LIN {X 0,Y 268.905,Z 288.913,A -85,B 0,C 180,E1 -18635.456,E2 -18635.456} C_VEL
LIN {X 0,Y 261.932,Z 271.443,A -85,B 0,C 180,E1 -18636.717,E2 -18636.717} C_VEL
LIN {X 0,Y 257.784,Z 261.083,A -85,B 0,C 180,E1 -18637.566,E2 -18637.566} C_VEL
LIN {X 0,Y 256.379,Z 255.314,A -85,B 0,C 180,E1 -18639.936,E2 -18639.936} C_VEL
LIN {X 0,Y 256.266,Z 255.064,A -85,B 0,C 180,E1 -18641.069,E2 -18641.069} C_VEL
LIN {X 0,Y 256.221,Z 255.067,A -85,B 0,C 180,E1 -18644.293,E2 -18644.293} C_VEL
LIN {X 0,Y 256.173,Z 255.073,A -85,B 0,C 180,E1 -18647.566,E2 -18647.566} C_VEL
LIN {X 0,Y 256.113,Z 255.08,A -85,B 0,C 180,E1 -18651.113,E2 -18651.113} C_VEL
LIN {X 0,Y 256.105,Z 255.077,A -85,B 0,C 180,E1 -18655.115,E2 -18655.115} C_VEL
LIN {X 0,Y 256.017,Z 255.078,A -85,B 0,C 180,E1 -18659.613,E2 -18659.613} C_VEL
LIN {X 0,Y 256.041,Z 255.087,A -85,B 0,C 180,E1 -18663.298,E2 -18663.298} C_VEL
LIN {X 0,Y 256.094,Z 255.082,A -85,B 0,C 180,E1 -18667.276,E2 -18667.276} C_VEL
LIN {X 0,Y 255.996,Z 255.082,A -85,B 0,C 180,E1 -18671.216,E2 -18671.216} C_VEL
LIN {X 0,Y 255.998,Z 255.094,A -85,B 0,C 180,E1 -18675.545,E2 -18675.545} C_VEL
LIN {X 0,Y 256,Z 255.085,A -85,B 0,C 180,E1 -18678.795,E2 -18678.795} C_VEL
LIN {X 0,Y 256.087,Z 255.063,A -85,B 0,C 180,E1 -18682.868,E2 -18682.868} C_VEL
LIN {X 0,Y 256.053,Z 255.09,A -85,B 0,C 180,E1 -18686.713,E2 -18686.713} C_VEL
LIN {X 0,Y 256.029,Z 255.058,A -85,B 0,C 180,E1 -18690.397,E2 -18690.397} C_VEL
LIN {X 0,Y 256.057,Z 255.074,A -85,B 0,C 180,E1 -18693.957,E2 -18693.957} C_VEL
LIN {X 0,Y 256.055,Z 255.089,A -85,B 0,C 180,E1 -18697.409,E2 -18697.409} C_VEL
LIN {X 0,Y 256.148,Z 255.047,A -85,B 0,C 180,E1 -18700.783,E2 -18700.783} C_VEL
LIN {X 0,Y 256.241,Z 255.032,A -85,B 0,C 180,E1 -18704.087,E2 -18704.087} C_VEL
LIN {X 0,Y 256.284,Z 255.057,A -85,B 0,C 180,E1 -18707.333,E2 -18707.333} C_VEL
LIN {X 0,Y 256.434,Z 255.031,A -85,B 0,C 180,E1 -18710.628,E2 -18710.628} C_VEL
LIN {X 0,Y 256.382,Z 255.005,A -85,B 0,C 180,E1 -18714.228,E2 -18714.228} C_VEL
LIN {X 0,Y 256.698,Z 255.005,A -85,B 0,C 180,E1 -18718.437,E2 -18718.437} C_VEL
LIN {X 0,Y 256.68,Z 255.005,A -85,B 0,C 180,E1 -18721.093,E2 -18721.093} C_VEL
LIN {X 0,Y 256.371,Z 255.041,A -85,B 0,C 180,E1 -18721.967,E2 -18721.967} C_VEL
LIN {X 0,Y 254.985,Z 255.205,A -85,B 0,C 180,E1 -18723.254,E2 -18723.254} C_VEL
LIN {X 0,Y 250.536,Z 255.744,A -85,B 0,C 180,E1 -18726.253,E2 -18726.253} C_VEL
LIN {X 0,Y 249.504,Z 255.89,A -85,B 0,C 180,E1 -18727.599,E2 -18727.599} C_VEL
LIN {X 0,Y 249.444,Z 255.899,A -85,B 0,C 180,E1 -18728.055,E2 -18728.055} C_VEL
LIN {X 0,Y 249.25,Z 255.935,A -85,B 0,C 180,E1 -18731.389,E2 -18731.389} C_VEL
LIN {X 0,Y 249.206,Z 255.915,A -85,B 0,C 180,E1 -18736.386,E2 -18736.386} C_VEL
LIN {X 0,Y 249.091,Z 255.95,A -85,B 0,C 180,E1 -18741.523,E2 -18741.523} C_VEL
LIN {X 0,Y 249.097,Z 255.938,A -85,B 0,C 180,E1 -18745.463,E2 -18745.463} C_VEL
LIN {X 0,Y 249.05,Z 255.959,A -85,B 0,C 180,E1 -18748.977,E2 -18748.977} C_VEL
LIN {X 0,Y 249.041,Z 255.95,A -85,B 0,C 180,E1 -18752.43,E2 -18752.43} C_VEL
LIN {X 0,Y 249.027,Z 255.956,A -85,B 0,C 180,E1 -18756.351,E2 -18756.351} C_VEL
LIN {X 0,Y 248.993,Z 255.969,A -85,B 0,C 180,E1 -18760.486,E2 -18760.486} C_VEL
LIN {X 0,Y 248.977,Z 255.972,A -85,B 0,C 180,E1 -18764.891,E2 -18764.891} C_VEL
LIN {X 0,Y 249.008,Z 255.964,A -85,B 0,C 180,E1 -18767.36,E2 -18767.36} C_VEL
LIN {X 0,Y 249.059,Z 255.959,A -85,B 0,C 180,E1 -18772.202,E2 -18772.202} C_VEL
LIN {X 0,Y 249.104,Z 255.988,A -85,B 0,C 180,E1 -18774.006,E2 -18774.006} C_VEL
LIN {X 0,Y 249.603,Z 258.24,A -85,B 0,C 180,E1 -18775.097,E2 -18775.097} C_VEL
LIN {X 0,Y 251.579,Z 267.236,A -85,B 0,C 180,E1 -18778.731,E2 -18778.731} C_VEL
LIN {X 0,Y 257.031,Z 280.617,A -85,B 0,C 180,E1 -18779.858,E2 -18779.858} C_VEL
LIN {X 0,Y 260.891,Z 291.121,A -85,B 0,C 180,E1 -18780.616,E2 -18780.616} C_VEL
LIN {X 0,Y 264.281,Z 312.794,A -85,B 0,C 180,E1 -18781.64,E2 -18781.64} C_VEL
LIN {X 0,Y 262.135,Z 374.903,A -85,B 0,C 180,E1 -18783.368,E2 -18783.368} C_VEL
LIN {X 0,Y 261.159,Z 388.066,A -85,B 0,C 180,E1 -18784.014,E2 -18784.014} C_VEL
LIN {X 0,Y 259.679,Z 401.335,A -85,B 0,C 180,E1 -18784.982,E2 -18784.982} C_VEL
LIN {X 0,Y 258.161,Z 412.517,A -85,B 0,C 180,E1 -18786.111,E2 -18786.111} C_VEL
LIN {X 0,Y 256.245,Z 424.145,A -85,B 0,C 180,E1 -18787.631,E2 -18787.631} C_VEL
LIN {X 0,Y 254.349,Z 434.623,A -85,B 0,C 180,E1 -18789.371,E2 -18789.371} C_VEL
LIN {X 0,Y 252.494,Z 444.866,A -85,B 0,C 180,E1 -18791.54,E2 -18791.54} C_VEL
LIN {X 0,Y 250.791,Z 453.135,A -85,B 0,C 180,E1 -18793.725,E2 -18793.725} C_VEL
LIN {X 0,Y 249.263,Z 460.448,A -85,B 0,C 180,E1 -18796.132,E2 -18796.132} C_VEL
LIN {X 0,Y 248.217,Z 466.292,A -85,B 0,C 180,E1 -18798.567,E2 -18798.567} C_VEL
LIN {X 0,Y 247.494,Z 470.875,A -85,B 0,C 180,E1 -18801.013,E2 -18801.013} C_VEL
LIN {X 0,Y 247.038,Z 474.348,A -85,B 0,C 180,E1 -18803.464,E2 -18803.464} C_VEL
LIN {X 0,Y 246.882,Z 476.113,A -85,B 0,C 180,E1 -18805.143,E2 -18805.143} C_VEL
LIN {X 0,Y 246.866,Z 478.303,A -85,B 0,C 180,E1 -18808.367,E2 -18808.367} C_VEL
LIN {X 0,Y 246.9,Z 478.807,A -85,B 0,C 180,E1 -18809.999,E2 -18809.999} C_VEL
LIN {X 0,Y 246.867,Z 478.878,A -85,B 0,C 180,E1 -18811.63,E2 -18811.63} C_VEL
LIN {X 0,Y 246.897,Z 477.862,A -85,B 0,C 180,E1 -18814.897,E2 -18814.897} C_VEL
LIN {X 0,Y 247.097,Z 476.762,A -85,B 0,C 180,E1 -18816.531,E2 -18816.531} C_VEL
LIN {X 0,Y 247.385,Z 475.213,A -85,B 0,C 180,E1 -18818.165,E2 -18818.165} C_VEL
LIN {X 0,Y 248.065,Z 472.112,A -85,B 0,C 180,E1 -18820.61,E2 -18820.61} C_VEL
LIN {X 0,Y 249.118,Z 467.968,A -85,B 0,C 180,E1 -18823.042,E2 -18823.042} C_VEL
LIN {X 0,Y 250.567,Z 462.667,A -85,B 0,C 180,E1 -18825.452,E2 -18825.452} C_VEL
LIN {X 0,Y 252.492,Z 456.034,A -85,B 0,C 180,E1 -18827.828,E2 -18827.828} C_VEL
LIN {X 0,Y 254.765,Z 447.424,A -85,B 0,C 180,E1 -18830.283,E2 -18830.283} C_VEL
LIN {X 0,Y 256.764,Z 439.438,A -85,B 0,C 180,E1 -18832.107,E2 -18832.107} C_VEL
LIN {X 0,Y 259.312,Z 429.101,A -85,B 0,C 180,E1 -18833.986,E2 -18833.986} C_VEL
LIN {X 0,Y 261.853,Z 417.489,A -85,B 0,C 180,E1 -18835.643,E2 -18835.643} C_VEL
LIN {X 0,Y 263.96,Z 405.99,A -85,B 0,C 180,E1 -18836.911,E2 -18836.911} C_VEL
LIN {X 0,Y 265.877,Z 392.843,A -85,B 0,C 180,E1 -18837.98,E2 -18837.98} C_VEL
LIN {X 0,Y 267.225,Z 380.531,A -85,B 0,C 180,E1 -18838.68,E2 -18838.68} C_VEL
LIN {X 0,Y 268.125,Z 367.233,A -85,B 0,C 180,E1 -18839.145,E2 -18839.145} C_VEL
LIN {X 0,Y 270.109,Z 314.39,A -85,B 0,C 180,E1 -18840.605,E2 -18840.605} C_VEL
LIN {X 0,Y 267.568,Z 298.937,A -85,B 0,C 180,E1 -18841.502,E2 -18841.502} C_VEL
LIN {X 0,Y 261.325,Z 284.682,A -85,B 0,C 180,E1 -18842.985,E2 -18842.985} C_VEL
LIN {X 0,Y 254.135,Z 270.585,A -85,B 0,C 180,E1 -18844.756,E2 -18844.756} C_VEL
LIN {X 0,Y 251.849,Z 266.387,A -85,B 0,C 180,E1 -18845.407,E2 -18845.407} C_VEL
LIN {X 0,Y 250.675,Z 261.826,A -85,B 0,C 180,E1 -18847.445,E2 -18847.445} C_VEL
LIN {X 0,Y 248.999,Z 256.011,A -85,B 0,C 180,E1 -18850.51,E2 -18850.51} C_VEL
LIN {X 0,Y 248.969,Z 255.972,A -85,B 0,C 180,E1 -18854.885,E2 -18854.885} C_VEL
LIN {X 0,Y 248.985,Z 255.971,A -85,B 0,C 180,E1 -18857.351,E2 -18857.351} C_VEL
LIN {X 0,Y 249.048,Z 255.957,A -85,B 0,C 180,E1 -18862.196,E2 -18862.196} C_VEL
LIN {X 0,Y 249.047,Z 255.957,A -85,B 0,C 180,E1 -18865.635,E2 -18865.635} C_VEL
LIN {X 0,Y 249.005,Z 255.962,A -85,B 0,C 180,E1 -18869.462,E2 -18869.462} C_VEL
LIN {X 0,Y 249.036,Z 255.954,A -85,B 0,C 180,E1 -18873.153,E2 -18873.153} C_VEL
LIN {X 0,Y 249.054,Z 255.95,A -85,B 0,C 180,E1 -18876.725,E2 -18876.725} C_VEL
LIN {X 0,Y 249.09,Z 255.955,A -85,B 0,C 180,E1 -18880.205,E2 -18880.205} C_VEL
LIN {X 0,Y 249.195,Z 255.944,A -85,B 0,C 180,E1 -18883.614,E2 -18883.614} C_VEL
LIN {X 0,Y 249.23,Z 255.938,A -85,B 0,C 180,E1 -18888.61,E2 -18888.61} C_VEL
LIN {X 0,Y 249.417,Z 255.903,A -85,B 0,C 180,E1 -18891.895,E2 -18891.895} C_VEL
LIN {X 0,Y 249.25,Z 255.93,A -85,B 0,C 180,E1 -18895.142,E2 -18895.142} C_VEL
LIN {X 0,Y 249.65,Z 255.887,A -85,B 0,C 180,E1 -18898.381,E2 -18898.381} C_VEL
LIN {X 0,Y 249.638,Z 255.877,A -85,B 0,C 180,E1 -18901.608,E2 -18901.608} C_VEL
LIN {X 0,Y 249.411,Z 255.909,A -85,B 0,C 180,E1 -18906.554,E2 -18906.554} C_VEL
LIN {X 0,Y 249.331,Z 255.918,A -85,B 0,C 180,E1 -18909.731,E2 -18909.731} C_VEL
LIN {X 0,Y 249.164,Z 255.947,A -85,B 0,C 180,E1 -18914.7,E2 -18914.7} C_VEL
LIN {X 0,Y 249.099,Z 255.954,A -85,B 0,C 180,E1 -18918.074,E2 -18918.074} C_VEL
LIN {X 0,Y 249.064,Z 255.962,A -85,B 0,C 180,E1 -18921.514,E2 -18921.514} C_VEL
LIN {X 0,Y 249.066,Z 255.957,A -85,B 0,C 180,E1 -18925.455,E2 -18925.455} C_VEL
LIN {X 0,Y 249.06,Z 256.056,A -85,B 0,C 180,E1 -18928.815,E2 -18928.815} C_VEL
LIN {X 0,Y 250.411,Z 261.075,A -85,B 0,C 180,E1 -18931.331,E2 -18931.331} C_VEL
LIN {X 0,Y 252.768,Z 265.242,A -85,B 0,C 180,E1 -18932.036,E2 -18932.036} C_VEL
LIN {X 0,Y 260.17,Z 278.693,A -85,B 0,C 180,E1 -18933.851,E2 -18933.851} C_VEL
LIN {X 0,Y 266.998,Z 293.384,A -85,B 0,C 180,E1 -18935.466,E2 -18935.466} C_VEL
LIN {X 0,Y 270.294,Z 301.89,A -85,B 0,C 180,E1 -18936.249,E2 -18936.249} C_VEL
LIN {X 0,Y 270.478,Z 305.292,A -85,B 0,C 180,E1 -18936.39,E2 -18936.39} C_VEL
LIN {X 0,Y 267.773,Z 368.475,A -85,B 0,C 180,E1 -18938.132,E2 -18938.132} C_VEL
LIN {X 0,Y 266.626,Z 381.328,A -85,B 0,C 180,E1 -18938.741,E2 -18938.741} C_VEL
LIN {X 0,Y 265.179,Z 393.57,A -85,B 0,C 180,E1 -18939.614,E2 -18939.614} C_VEL
LIN {X 0,Y 263.303,Z 405.552,A -85,B 0,C 180,E1 -18940.769,E2 -18940.769} C_VEL
LIN {X 0,Y 260.997,Z 417.533,A -85,B 0,C 180,E1 -18942.305,E2 -18942.305} C_VEL
LIN {X 0,Y 258.672,Z 427.674,A -85,B 0,C 180,E1 -18943.948,E2 -18943.948} C_VEL
LIN {X 0,Y 256.398,Z 436.734,A -85,B 0,C 180,E1 -18945.78,E2 -18945.78} C_VEL
LIN {X 0,Y 254.141,Z 445.083,A -85,B 0,C 180,E1 -18947.888,E2 -18947.888} C_VEL
LIN {X 0,Y 252.228,Z 452.224,A -85,B 0,C 180,E1 -18950.146,E2 -18950.146} C_VEL
LIN {X 0,Y 250.271,Z 459.008,A -85,B 0,C 180,E1 -18952.863,E2 -18952.863} C_VEL
LIN {X 0,Y 248.792,Z 464.189,A -85,B 0,C 180,E1 -18955.602,E2 -18955.602} C_VEL
LIN {X 0,Y 247.8,Z 467.877,A -85,B 0,C 180,E1 -18958.29,E2 -18958.29} C_VEL
LIN {X 0,Y 247.073,Z 470.447,A -85,B 0,C 180,E1 -18961.083,E2 -18961.083} C_VEL
LIN {X 0,Y 246.731,Z 471.477,A -85,B 0,C 180,E1 -18962.888,E2 -18962.888} C_VEL
LIN {X 0,Y 246.46,Z 472.111,A -85,B 0,C 180,E1 -18965.836,E2 -18965.836} C_VEL
LIN {X 0,Y 246.446,Z 471.646,A -85,B 0,C 180,E1 -18968.241,E2 -18968.241} C_VEL
LIN {X 0,Y 246.573,Z 470.671,A -85,B 0,C 180,E1 -18970.129,E2 -18970.129} C_VEL
LIN {X 0,Y 246.773,Z 469.404,A -85,B 0,C 180,E1 -18971.745,E2 -18971.745} C_VEL
LIN {X 0,Y 247.075,Z 467.612,A -85,B 0,C 180,E1 -18973.476,E2 -18973.476} C_VEL
LIN {X 0,Y 247.703,Z 463.988,A -85,B 0,C 180,E1 -18976.046,E2 -18976.046} C_VEL
LIN {X 0,Y 248.568,Z 459.181,A -85,B 0,C 180,E1 -18978.586,E2 -18978.586} C_VEL
LIN {X 0,Y 249.801,Z 452.76,A -85,B 0,C 180,E1 -18981.198,E2 -18981.198} C_VEL
LIN {X 0,Y 251.326,Z 445.351,A -85,B 0,C 180,E1 -18983.579,E2 -18983.579} C_VEL
LIN {X 0,Y 252.879,Z 437.663,A -85,B 0,C 180,E1 -18985.576,E2 -18985.576} C_VEL
LIN {X 0,Y 254.781,Z 427.879,A -85,B 0,C 180,E1 -18987.63,E2 -18987.63} C_VEL
LIN {X 0,Y 256.709,Z 417.119,A -85,B 0,C 180,E1 -18989.413,E2 -18989.413} C_VEL
LIN {X 0,Y 258.635,Z 405.096,A -85,B 0,C 180,E1 -18990.974,E2 -18990.974} C_VEL
LIN {X 0,Y 259.987,Z 394.162,A -85,B 0,C 180,E1 -18992.07,E2 -18992.07} C_VEL
LIN {X 0,Y 261.32,Z 381.02,A -85,B 0,C 180,E1 -18993.033,E2 -18993.033} C_VEL
LIN {X 0,Y 262.303,Z 367.755,A -85,B 0,C 180,E1 -18993.676,E2 -18993.676} C_VEL
LIN {X 0,Y 264.475,Z 300.673,A -85,B 0,C 180,E1 -18995.549,E2 -18995.549} C_VEL
LIN {X 0,Y 262.663,Z 291.146,A -85,B 0,C 180,E1 -18996.03,E2 -18996.03} C_VEL
LIN {X 0,Y 253.003,Z 266.946,A -85,B 0,C 180,E1 -18997.875,E2 -18997.875} C_VEL
LIN {X 0,Y 250.54,Z 261.15,A -85,B 0,C 180,E1 -18998.419,E2 -18998.419} C_VEL
LIN {X 0,Y 249.293,Z 256.147,A -85,B 0,C 180,E1 -19000.559,E2 -19000.559} C_VEL
LIN {X 0,Y 249.167,Z 255.949,A -85,B 0,C 180,E1 -19004.707,E2 -19004.707} C_VEL
LIN {X 0,Y 249.104,Z 255.957,A -85,B 0,C 180,E1 -19008.081,E2 -19008.081} C_VEL
LIN {X 0,Y 249.052,Z 255.961,A -85,B 0,C 180,E1 -19011.523,E2 -19011.523} C_VEL
LIN {X 0,Y 249.057,Z 255.957,A -85,B 0,C 180,E1 -19015.463,E2 -19015.463} C_VEL
LIN {X 0,Y 249.002,Z 255.952,A -85,B 0,C 180,E1 -19018.974,E2 -19018.974} C_VEL
LIN {X 0,Y 249.001,Z 255.969,A -85,B 0,C 180,E1 -19022.431,E2 -19022.431} C_VEL
LIN {X 0,Y 248.99,Z 255.954,A -85,B 0,C 180,E1 -19026.353,E2 -19026.353} C_VEL
LIN {X 0,Y 248.957,Z 255.964,A -85,B 0,C 180,E1 -19030.489,E2 -19030.489} C_VEL
LIN {X 0,Y 248.943,Z 255.967,A -85,B 0,C 180,E1 -19034.894,E2 -19034.894} C_VEL
LIN {X 0,Y 248.975,Z 255.969,A -85,B 0,C 180,E1 -19037.363,E2 -19037.363} C_VEL
LIN {X 0,Y 249.028,Z 255.936,A -85,B 0,C 180,E1 -19042.206,E2 -19042.206} C_VEL
LIN {X 0,Y 249.029,Z 255.964,A -85,B 0,C 180,E1 -19045.645,E2 -19045.645} C_VEL
LIN {X 0,Y 248.982,Z 255.946,A -85,B 0,C 180,E1 -19049.471,E2 -19049.471} C_VEL
LIN {X 0,Y 249.004,Z 255.942,A -85,B 0,C 180,E1 -19053.161,E2 -19053.161} C_VEL
LIN {X 0,Y 249.001,Z 255.967,A -85,B 0,C 180,E1 -19056.732,E2 -19056.732} C_VEL
LIN {X 0,Y 249.076,Z 255.937,A -85,B 0,C 180,E1 -19060.215,E2 -19060.215} C_VEL
LIN {X 0,Y 249.192,Z 255.904,A -85,B 0,C 180,E1 -19063.625,E2 -19063.625} C_VEL
LIN {X 0,Y 249.24,Z 255.936,A -85,B 0,C 180,E1 -19068.622,E2 -19068.622} C_VEL
LIN {X 0,Y 249.417,Z 255.889,A -85,B 0,C 180,E1 -19071.907,E2 -19071.907} C_VEL
LIN {X 0,Y 249.261,Z 255.897,A -85,B 0,C 180,E1 -19075.153,E2 -19075.153} C_VEL
LIN {X 0,Y 249.659,Z 255.881,A -85,B 0,C 180,E1 -19078.392,E2 -19078.392} C_VEL
LIN {X 0,Y 249.662,Z 255.879,A -85,B 0,C 180,E1 -19081.619,E2 -19081.619} C_VEL
LIN {X 0,Y 249.441,Z 255.88,A -85,B 0,C 180,E1 -19086.476,E2 -19086.476} C_VEL
LIN {X 0,Y 249.444,Z 255.899,A -85,B 0,C 180,E1 -19088.055,E2 -19088.055} C_VEL
LIN {X 0,Y 249.171,Z 255.947,A -85,B 0,C 180,E1 -19088.954,E2 -19088.954} C_VEL
LIN {X 0,Y 247.836,Z 256.118,A -85,B 0,C 180,E1 -19090.282,E2 -19090.282} C_VEL
LIN {X 0,Y 243.384,Z 256.651,A -85,B 0,C 180,E1 -19093.372,E2 -19093.372} C_VEL
LIN {X 0,Y 242.253,Z 256.777,A -85,B 0,C 180,E1 -19094.758,E2 -19094.758} C_VEL
LIN {X 0,Y 242.14,Z 256.789,A -85,B 0,C 180,E1 -19095.229,E2 -19095.229} C_VEL
LIN {X 0,Y 242.06,Z 256.828,A -85,B 0,C 180,E1 -19098.63,E2 -19098.63} C_VEL
LIN {X 0,Y 242.014,Z 256.825,A -85,B 0,C 180,E1 -19102.185,E2 -19102.185} C_VEL
LIN {X 0,Y 242.045,Z 256.821,A -85,B 0,C 180,E1 -19105.825,E2 -19105.825} C_VEL
LIN {X 0,Y 241.982,Z 256.834,A -85,B 0,C 180,E1 -19109.592,E2 -19109.592} C_VEL
LIN {X 0,Y 241.993,Z 256.837,A -85,B 0,C 180,E1 -19113.496,E2 -19113.496} C_VEL
LIN {X 0,Y 241.997,Z 256.826,A -85,B 0,C 180,E1 -19117.586,E2 -19117.586} C_VEL
LIN {X 0,Y 241.922,Z 256.838,A -85,B 0,C 180,E1 -19121.931,E2 -19121.931} C_VEL
LIN {X 0,Y 241.924,Z 256.843,A -85,B 0,C 180,E1 -19126.58,E2 -19126.58} C_VEL
LIN {X 0,Y 242.009,Z 256.837,A -85,B 0,C 180,E1 -19131.643,E2 -19131.643} C_VEL
LIN {X 0,Y 242.111,Z 257.081,A -85,B 0,C 180,E1 -19133.569,E2 -19133.569} C_VEL
LIN {X 0,Y 244.107,Z 266.267,A -85,B 0,C 180,E1 -19137.558,E2 -19137.558} C_VEL
LIN {X 0,Y 244.397,Z 267.469,A -85,B 0,C 180,E1 -19137.888,E2 -19137.888} C_VEL
LIN {X 0,Y 250.889,Z 282.886,A -85,B 0,C 180,E1 -19139.224,E2 -19139.224} C_VEL
LIN {X 0,Y 254.852,Z 294.015,A -85,B 0,C 180,E1 -19140.041,E2 -19140.041} C_VEL
LIN {X 0,Y 257.856,Z 313.922,A -85,B 0,C 180,E1 -19141.004,E2 -19141.004} C_VEL
LIN {X 0,Y 255.629,Z 375.004,A -85,B 0,C 180,E1 -19142.745,E2 -19142.745} C_VEL
LIN {X 0,Y 254.632,Z 388.103,A -85,B 0,C 180,E1 -19143.406,E2 -19143.406} C_VEL
LIN {X 0,Y 253.094,Z 401.332,A -85,B 0,C 180,E1 -19144.395,E2 -19144.395} C_VEL
LIN {X 0,Y 251.383,Z 413.285,A -85,B 0,C 180,E1 -19145.645,E2 -19145.645} C_VEL
LIN {X 0,Y 249.423,Z 424.76,A -85,B 0,C 180,E1 -19147.204,E2 -19147.204} C_VEL
LIN {X 0,Y 247.469,Z 435.111,A -85,B 0,C 180,E1 -19148.988,E2 -19148.988} C_VEL
LIN {X 0,Y 245.57,Z 445.164,A -85,B 0,C 180,E1 -19151.201,E2 -19151.201} C_VEL
LIN {X 0,Y 243.685,Z 454.101,A -85,B 0,C 180,E1 -19153.667,E2 -19153.667} C_VEL
LIN {X 0,Y 242.146,Z 461.181,A -85,B 0,C 180,E1 -19156.145,E2 -19156.145} C_VEL
LIN {X 0,Y 240.923,Z 467.649,A -85,B 0,C 180,E1 -19159.069,E2 -19159.069} C_VEL
LIN {X 0,Y 240.253,Z 471.894,A -85,B 0,C 180,E1 -19161.588,E2 -19161.588} C_VEL
LIN {X 0,Y 239.978,Z 474.14,A -85,B 0,C 180,E1 -19163.271,E2 -19163.271} C_VEL
LIN {X 0,Y 239.777,Z 476.188,A -85,B 0,C 180,E1 -19165.291,E2 -19165.291} C_VEL
LIN {X 0,Y 239.78,Z 478.16,A -85,B 0,C 180,E1 -19168.319,E2 -19168.319} C_VEL
LIN {X 0,Y 239.813,Z 478.694,A -85,B 0,C 180,E1 -19169.999,E2 -19169.999} C_VEL
LIN {X 0,Y 239.78,Z 478.788,A -85,B 0,C 180,E1 -19171.678,E2 -19171.678} C_VEL
LIN {X 0,Y 239.817,Z 477.808,A -85,B 0,C 180,E1 -19175.042,E2 -19175.042} C_VEL
LIN {X 0,Y 240.045,Z 476.737,A -85,B 0,C 180,E1 -19176.724,E2 -19176.724} C_VEL
LIN {X 0,Y 240.34,Z 475.218,A -85,B 0,C 180,E1 -19178.406,E2 -19178.406} C_VEL
LIN {X 0,Y 241.062,Z 472.163,A -85,B 0,C 180,E1 -19180.922,E2 -19180.922} C_VEL
LIN {X 0,Y 242.172,Z 468.065,A -85,B 0,C 180,E1 -19183.423,E2 -19183.423} C_VEL
LIN {X 0,Y 244.068,Z 461.802,A -85,B 0,C 180,E1 -19186.304,E2 -19186.304} C_VEL
LIN {X 0,Y 246.159,Z 454.998,A -85,B 0,C 180,E1 -19188.734,E2 -19188.734} C_VEL
LIN {X 0,Y 248.398,Z 446.621,A -85,B 0,C 180,E1 -19191.126,E2 -19191.126} C_VEL
LIN {X 0,Y 250.702,Z 437.883,A -85,B 0,C 180,E1 -19193.106,E2 -19193.106} C_VEL
LIN {X 0,Y 253.452,Z 427.226,A -85,B 0,C 180,E1 -19195.014,E2 -19195.014} C_VEL
LIN {X 0,Y 255.775,Z 416.676,A -85,B 0,C 180,E1 -19196.518,E2 -19196.518} C_VEL
LIN {X 0,Y 258.027,Z 404.923,A -85,B 0,C 180,E1 -19197.802,E2 -19197.802} C_VEL
LIN {X 0,Y 259.851,Z 392.794,A -85,B 0,C 180,E1 -19198.799,E2 -19198.799} C_VEL
LIN {X 0,Y 261.26,Z 380.489,A -85,B 0,C 180,E1 -19199.512,E2 -19199.512} C_VEL
LIN {X 0,Y 262.197,Z 366.8,A -85,B 0,C 180,E1 -19200,E2 -19200} C_VEL
LIN {X 0,Y 264.279,Z 315.513,A -85,B 0,C 180,E1 -19201.438,E2 -19201.438} C_VEL
LIN {X 0,Y 262.003,Z 301.708,A -85,B 0,C 180,E1 -19202.274,E2 -19202.274} C_VEL
LIN {X 0,Y 256.332,Z 288.59,A -85,B 0,C 180,E1 -19203.69,E2 -19203.69} C_VEL
LIN {X 0,Y 249.293,Z 274.721,A -85,B 0,C 180,E1 -19205.504,E2 -19205.504} C_VEL
LIN {X 0,Y 244.666,Z 266.307,A -85,B 0,C 180,E1 -19206.839,E2 -19206.839} C_VEL
LIN {X 0,Y 243.499,Z 262.145,A -85,B 0,C 180,E1 -19208.798,E2 -19208.798} C_VEL
LIN {X 0,Y 241.959,Z 256.871,A -85,B 0,C 180,E1 -19211.778,E2 -19211.778} C_VEL
LIN {X 0,Y 241.907,Z 256.851,A -85,B 0,C 180,E1 -19216.576,E2 -19216.576} C_VEL
LIN {X 0,Y 241.999,Z 256.833,A -85,B 0,C 180,E1 -19221.637,E2 -19221.637} C_VEL
LIN {X 0,Y 241.978,Z 256.836,A -85,B 0,C 180,E1 -19224.482,E2 -19224.482} C_VEL
LIN {X 0,Y 241.956,Z 256.837,A -85,B 0,C 180,E1 -19228.472,E2 -19228.472} C_VEL
LIN {X 0,Y 241.969,Z 256.834,A -85,B 0,C 180,E1 -19232.303,E2 -19232.303} C_VEL
LIN {X 0,Y 242.025,Z 256.83,A -85,B 0,C 180,E1 -19236.007,E2 -19236.007} C_VEL
LIN {X 0,Y 242.024,Z 256.837,A -85,B 0,C 180,E1 -19239.601,E2 -19239.601} C_VEL
LIN {X 0,Y 242.127,Z 256.82,A -85,B 0,C 180,E1 -19243.301,E2 -19243.301} C_VEL
LIN {X 0,Y 242.164,Z 256.818,A -85,B 0,C 180,E1 -19248.273,E2 -19248.273} C_VEL
LIN {X 0,Y 242.37,Z 256.78,A -85,B 0,C 180,E1 -19251.658,E2 -19251.658} C_VEL
LIN {X 0,Y 242.395,Z 256.789,A -85,B 0,C 180,E1 -19253.335,E2 -19253.335} C_VEL
LIN {X 0,Y 242.609,Z 256.764,A -85,B 0,C 180,E1 -19258.334,E2 -19258.334} C_VEL
LIN {X 0,Y 242.597,Z 256.754,A -85,B 0,C 180,E1 -19261.654,E2 -19261.654} C_VEL
LIN {X 0,Y 242.388,Z 256.786,A -85,B 0,C 180,E1 -19266.654,E2 -19266.654} C_VEL
LIN {X 0,Y 242.254,Z 256.8,A -85,B 0,C 180,E1 -19270.018,E2 -19270.018} C_VEL
LIN {X 0,Y 242.122,Z 256.827,A -85,B 0,C 180,E1 -19275.137,E2 -19275.137} C_VEL
LIN {X 0,Y 242.036,Z 256.839,A -85,B 0,C 180,E1 -19278.62,E2 -19278.62} C_VEL
LIN {X 0,Y 241.986,Z 256.84,A -85,B 0,C 180,E1 -19282.176,E2 -19282.176} C_VEL
LIN {X 0,Y 242.014,Z 256.836,A -85,B 0,C 180,E1 -19285.816,E2 -19285.816} C_VEL
LIN {X 0,Y 241.987,Z 257.057,A -85,B 0,C 180,E1 -19287.683,E2 -19287.683} C_VEL
LIN {X 0,Y 243.174,Z 261.208,A -85,B 0,C 180,E1 -19289.836,E2 -19289.836} C_VEL
LIN {X 0,Y 245.634,Z 265.496,A -85,B 0,C 180,E1 -19290.633,E2 -19290.633} C_VEL
LIN {X 0,Y 251.458,Z 275.598,A -85,B 0,C 180,E1 -19292.184,E2 -19292.184} C_VEL
LIN {X 0,Y 257.189,Z 286.722,A -85,B 0,C 180,E1 -19293.634,E2 -19293.634} C_VEL
LIN {X 0,Y 263.401,Z 300.875,A -85,B 0,C 180,E1 -19295.163,E2 -19295.163} C_VEL
LIN {X 0,Y 264.646,Z 304.114,A -85,B 0,C 180,E1 -19295.469,E2 -19295.469} C_VEL
LIN {X 0,Y 261.905,Z 367.933,A -85,B 0,C 180,E1 -19297.272,E2 -19297.272} C_VEL
LIN {X 0,Y 260.704,Z 380.858,A -85,B 0,C 180,E1 -19297.877,E2 -19297.877} C_VEL
LIN {X 0,Y 259.163,Z 393.357,A -85,B 0,C 180,E1 -19298.775,E2 -19298.775} C_VEL
LIN {X 0,Y 257.418,Z 404.341,A -85,B 0,C 180,E1 -19299.84,E2 -19299.84} C_VEL
LIN {X 0,Y 255.282,Z 415.217,A -85,B 0,C 180,E1 -19301.192,E2 -19301.192} C_VEL
LIN {X 0,Y 252.868,Z 425.724,A -85,B 0,C 180,E1 -19302.86,E2 -19302.86} C_VEL
LIN {X 0,Y 250.197,Z 435.884,A -85,B 0,C 180,E1 -19304.888,E2 -19304.888} C_VEL
LIN {X 0,Y 247.754,Z 444.636,A -85,B 0,C 180,E1 -19307.096,E2 -19307.096} C_VEL
LIN {X 0,Y 245.669,Z 451.868,A -85,B 0,C 180,E1 -19309.399,E2 -19309.399} C_VEL
LIN {X 0,Y 243.789,Z 457.87,A -85,B 0,C 180,E1 -19311.782,E2 -19311.782} C_VEL
LIN {X 0,Y 242.18,Z 463.22,A -85,B 0,C 180,E1 -19314.524,E2 -19314.524} C_VEL
LIN {X 0,Y 241.352,Z 466.115,A -85,B 0,C 180,E1 -19316.411,E2 -19316.411} C_VEL
LIN {X 0,Y 240.687,Z 468.362,A -85,B 0,C 180,E1 -19318.294,E2 -19318.294} C_VEL
LIN {X 0,Y 239.893,Z 471,A -85,B 0,C 180,E1 -19321.493,E2 -19321.493} C_VEL
LIN {X 0,Y 239.479,Z 471.975,A -85,B 0,C 180,E1 -19323.885,E2 -19323.885} C_VEL
LIN {X 0,Y 239.37,Z 472.21,A -85,B 0,C 180,E1 -19325.731,E2 -19325.731} C_VEL
LIN {X 0,Y 239.319,Z 471.928,A -85,B 0,C 180,E1 -19327.559,E2 -19327.559} C_VEL
LIN {X 0,Y 239.445,Z 470.923,A -85,B 0,C 180,E1 -19329.902,E2 -19329.902} C_VEL
LIN {X 0,Y 239.885,Z 468.364,A -85,B 0,C 180,E1 -19332.966,E2 -19332.966} C_VEL
LIN {X 0,Y 240.492,Z 464.931,A -85,B 0,C 180,E1 -19335.655,E2 -19335.655} C_VEL
LIN {X 0,Y 241.296,Z 460.466,A -85,B 0,C 180,E1 -19338.237,E2 -19338.237} C_VEL
LIN {X 0,Y 242.594,Z 454.074,A -85,B 0,C 180,E1 -19341.068,E2 -19341.068} C_VEL
LIN {X 0,Y 244.312,Z 445.966,A -85,B 0,C 180,E1 -19343.809,E2 -19343.809} C_VEL
LIN {X 0,Y 246.163,Z 437.135,A -85,B 0,C 180,E1 -19346.168,E2 -19346.168} C_VEL
LIN {X 0,Y 248.073,Z 427.673,A -85,B 0,C 180,E1 -19348.175,E2 -19348.175} C_VEL
LIN {X 0,Y 250.08,Z 416.846,A -85,B 0,C 180,E1 -19350.001,E2 -19350.001} C_VEL
LIN {X 0,Y 252.058,Z 404.714,A -85,B 0,C 180,E1 -19351.599,E2 -19351.599} C_VEL
LIN {X 0,Y 253.665,Z 391.883,A -85,B 0,C 180,E1 -19352.868,E2 -19352.868} C_VEL
LIN {X 0,Y 254.906,Z 379.464,A -85,B 0,C 180,E1 -19353.756,E2 -19353.756} C_VEL
LIN {X 0,Y 255.843,Z 367.049,A -85,B 0,C 180,E1 -19354.334,E2 -19354.334} C_VEL
LIN {X 0,Y 258.14,Z 302.188,A -85,B 0,C 180,E1 -19356.169,E2 -19356.169} C_VEL
LIN {X 0,Y 256.535,Z 293.573,A -85,B 0,C 180,E1 -19356.616,E2 -19356.616} C_VEL
LIN {X 0,Y 246.263,Z 267.878,A -85,B 0,C 180,E1 -19358.668,E2 -19358.668} C_VEL
LIN {X 0,Y 243.281,Z 261.249,A -85,B 0,C 180,E1 -19359.328,E2 -19359.328} C_VEL
LIN {X 0,Y 242.197,Z 256.901,A -85,B 0,C 180,E1 -19361.296,E2 -19361.296} C_VEL
LIN {X 0,Y 242.127,Z 256.825,A -85,B 0,C 180,E1 -19365.145,E2 -19365.145} C_VEL
LIN {X 0,Y 242.037,Z 256.835,A -85,B 0,C 180,E1 -19368.628,E2 -19368.628} C_VEL
LIN {X 0,Y 241.975,Z 256.844,A -85,B 0,C 180,E1 -19372.185,E2 -19372.185} C_VEL
LIN {X 0,Y 242.007,Z 256.837,A -85,B 0,C 180,E1 -19375.825,E2 -19375.825} C_VEL
LIN {X 0,Y 241.939,Z 256.831,A -85,B 0,C 180,E1 -19379.594,E2 -19379.594} C_VEL
LIN {X 0,Y 241.955,Z 256.839,A -85,B 0,C 180,E1 -19383.498,E2 -19383.498} C_VEL
LIN {X 0,Y 241.962,Z 256.842,A -85,B 0,C 180,E1 -19387.588,E2 -19387.588} C_VEL
LIN {X 0,Y 241.887,Z 256.831,A -85,B 0,C 180,E1 -19391.935,E2 -19391.935} C_VEL
LIN {X 0,Y 241.89,Z 256.855,A -85,B 0,C 180,E1 -19396.584,E2 -19396.584} C_VEL
LIN {X 0,Y 241.978,Z 256.81,A -85,B 0,C 180,E1 -19401.647,E2 -19401.647} C_VEL
LIN {X 0,Y 241.96,Z 256.838,A -85,B 0,C 180,E1 -19404.493,E2 -19404.493} C_VEL
LIN {X 0,Y 241.936,Z 256.834,A -85,B 0,C 180,E1 -19408.482,E2 -19408.482} C_VEL
LIN {X 0,Y 241.941,Z 256.812,A -85,B 0,C 180,E1 -19412.312,E2 -19412.312} C_VEL
LIN {X 0,Y 241.975,Z 256.842,A -85,B 0,C 180,E1 -19416.014,E2 -19416.014} C_VEL
LIN {X 0,Y 242.012,Z 256.821,A -85,B 0,C 180,E1 -19419.612,E2 -19419.612} C_VEL
LIN {X 0,Y 242.112,Z 256.782,A -85,B 0,C 180,E1 -19423.322,E2 -19423.322} C_VEL
LIN {X 0,Y 242.148,Z 256.816,A -85,B 0,C 180,E1 -19426.58,E2 -19426.58} C_VEL
LIN {X 0,Y 242.342,Z 256.787,A -85,B 0,C 180,E1 -19430.411,E2 -19430.411} C_VEL
LIN {X 0,Y 242.396,Z 256.748,A -85,B 0,C 180,E1 -19433.346,E2 -19433.346} C_VEL
LIN {X 0,Y 242.619,Z 256.757,A -85,B 0,C 180,E1 -19438.346,E2 -19438.346} C_VEL
LIN {X 0,Y 242.621,Z 256.754,A -85,B 0,C 180,E1 -19441.666,E2 -19441.666} C_VEL
LIN {X 0,Y 242.413,Z 256.756,A -85,B 0,C 180,E1 -19446.665,E2 -19446.665} C_VEL
LIN {X 0,Y 242.275,Z 256.805,A -85,B 0,C 180,E1 -19450.029,E2 -19450.029} C_VEL
LIN {X 0,Y 242.146,Z 256.788,A -85,B 0,C 180,E1 -19455.147,E2 -19455.147} C_VEL
LIN {X 0,Y 242.14,Z 256.789,A -85,B 0,C 180,E1 -19455.229,E2 -19455.229} C_VEL
LIN {X 0,Y 241.416,Z 256.887,A -85,B 0,C 180,E1 -19456.615,E2 -19456.615} C_VEL
LIN {X 0,Y 238.537,Z 257.269,A -85,B 0,C 180,E1 -19458.876,E2 -19458.876} C_VEL
LIN {X 0,Y 236.112,Z 257.573,A -85,B 0,C 180,E1 -19460.718,E2 -19460.718} C_VEL
LIN {X 0,Y 235.058,Z 257.691,A -85,B 0,C 180,E1 -19462.148,E2 -19462.148} C_VEL
LIN {X 0,Y 234.963,Z 257.696,A -85,B 0,C 180,E1 -19462.632,E2 -19462.632} C_VEL
LIN {X 0,Y 234.958,Z 257.712,A -85,B 0,C 180,E1 -19466.664,E2 -19466.664} C_VEL
LIN {X 0,Y 234.912,Z 257.706,A -85,B 0,C 180,E1 -19470.576,E2 -19470.576} C_VEL
LIN {X 0,Y 234.936,Z 257.721,A -85,B 0,C 180,E1 -19474.643,E2 -19474.643} C_VEL
LIN {X 0,Y 234.927,Z 257.716,A -85,B 0,C 180,E1 -19478.938,E2 -19478.938} C_VEL
LIN {X 0,Y 234.868,Z 257.72,A -85,B 0,C 180,E1 -19483.497,E2 -19483.497} C_VEL
LIN {X 0,Y 234.876,Z 257.721,A -85,B 0,C 180,E1 -19486.51,E2 -19486.51} C_VEL
LIN {X 0,Y 234.934,Z 257.721,A -85,B 0,C 180,E1 -19491.08,E2 -19491.08} C_VEL
LIN {X 0,Y 235.01,Z 257.905,A -85,B 0,C 180,E1 -19492.862,E2 -19492.862} C_VEL
LIN {X 0,Y 237.051,Z 266.878,A -85,B 0,C 180,E1 -19496.86,E2 -19496.86} C_VEL
LIN {X 0,Y 239.02,Z 271.789,A -85,B 0,C 180,E1 -19497.382,E2 -19497.382} C_VEL
LIN {X 0,Y 245.416,Z 287.03,A -85,B 0,C 180,E1 -19498.712,E2 -19498.712} C_VEL
LIN {X 0,Y 248.602,Z 295.669,A -85,B 0,C 180,E1 -19499.383,E2 -19499.383} C_VEL
LIN {X 0,Y 251.421,Z 314.252,A -85,B 0,C 180,E1 -19500.32,E2 -19500.32} C_VEL
LIN {X 0,Y 249.163,Z 374.852,A -85,B 0,C 180,E1 -19502.091,E2 -19502.091} C_VEL
LIN {X 0,Y 248.108,Z 387.96,A -85,B 0,C 180,E1 -19502.763,E2 -19502.763} C_VEL
LIN {X 0,Y 246.523,Z 401.2,A -85,B 0,C 180,E1 -19503.775,E2 -19503.775} C_VEL
LIN {X 0,Y 244.894,Z 412.369,A -85,B 0,C 180,E1 -19504.956,E2 -19504.956} C_VEL
LIN {X 0,Y 242.883,Z 423.997,A -85,B 0,C 180,E1 -19506.554,E2 -19506.554} C_VEL
LIN {X 0,Y 240.786,Z 434.465,A -85,B 0,C 180,E1 -19508.376,E2 -19508.376} C_VEL
LIN {X 0,Y 239.006,Z 443.72,A -85,B 0,C 180,E1 -19510.413,E2 -19510.413} C_VEL
LIN {X 0,Y 237.075,Z 452.288,A -85,B 0,C 180,E1 -19512.754,E2 -19512.754} C_VEL
LIN {X 0,Y 235.449,Z 459.722,A -85,B 0,C 180,E1 -19515.301,E2 -19515.301} C_VEL
LIN {X 0,Y 234.267,Z 465.677,A -85,B 0,C 180,E1 -19517.876,E2 -19517.876} C_VEL
LIN {X 0,Y 233.43,Z 470.36,A -85,B 0,C 180,E1 -19520.467,E2 -19520.467} C_VEL
LIN {X 0,Y 232.912,Z 473.912,A -85,B 0,C 180,E1 -19523.066,E2 -19523.066} C_VEL
LIN {X 0,Y 232.689,Z 476.216,A -85,B 0,C 180,E1 -19525.403,E2 -19525.403} C_VEL
LIN {X 0,Y 232.676,Z 478.013,A -85,B 0,C 180,E1 -19528.268,E2 -19528.268} C_VEL
LIN {X 0,Y 232.728,Z 478.572,A -85,B 0,C 180,E1 -19529.999,E2 -19529.999} C_VEL
LIN {X 0,Y 232.677,Z 478.699,A -85,B 0,C 180,E1 -19531.729,E2 -19531.729} C_VEL
LIN {X 0,Y 232.748,Z 477.758,A -85,B 0,C 180,E1 -19535.196,E2 -19535.196} C_VEL
LIN {X 0,Y 232.99,Z 476.71,A -85,B 0,C 180,E1 -19536.929,E2 -19536.929} C_VEL
LIN {X 0,Y 233.294,Z 475.229,A -85,B 0,C 180,E1 -19538.662,E2 -19538.662} C_VEL
LIN {X 0,Y 234.068,Z 472.216,A -85,B 0,C 180,E1 -19541.253,E2 -19541.253} C_VEL
LIN {X 0,Y 235.239,Z 468.162,A -85,B 0,C 180,E1 -19543.826,E2 -19543.826} C_VEL
LIN {X 0,Y 237.25,Z 461.947,A -85,B 0,C 180,E1 -19546.786,E2 -19546.786} C_VEL
LIN {X 0,Y 239.44,Z 455.202,A -85,B 0,C 180,E1 -19549.28,E2 -19549.28} C_VEL
LIN {X 0,Y 241.709,Z 447.223,A -85,B 0,C 180,E1 -19551.655,E2 -19551.655} C_VEL
LIN {X 0,Y 244.218,Z 438.302,A -85,B 0,C 180,E1 -19553.757,E2 -19553.757} C_VEL
LIN {X 0,Y 247.075,Z 427.766,A -85,B 0,C 180,E1 -19555.706,E2 -19555.706} C_VEL
LIN {X 0,Y 249.489,Z 417.353,A -85,B 0,C 180,E1 -19557.241,E2 -19557.241} C_VEL
LIN {X 0,Y 251.817,Z 405.897,A -85,B 0,C 180,E1 -19558.549,E2 -19558.549} C_VEL
LIN {X 0,Y 253.687,Z 394.098,A -85,B 0,C 180,E1 -19559.567,E2 -19559.567} C_VEL
LIN {X 0,Y 255.264,Z 381.205,A -85,B 0,C 180,E1 -19560.35,E2 -19560.35} C_VEL
LIN {X 0,Y 256.246,Z 369.089,A -85,B 0,C 180,E1 -19560.812,E2 -19560.812} C_VEL
LIN {X 0,Y 258.491,Z 317.147,A -85,B 0,C 180,E1 -19562.294,E2 -19562.294} C_VEL
LIN {X 0,Y 256.509,Z 304.413,A -85,B 0,C 180,E1 -19563.08,E2 -19563.08} C_VEL
LIN {X 0,Y 250.351,Z 290.281,A -85,B 0,C 180,E1 -19564.708,E2 -19564.708} C_VEL
LIN {X 0,Y 244.555,Z 278.916,A -85,B 0,C 180,E1 -19566.286,E2 -19566.286} C_VEL
LIN {X 0,Y 239.19,Z 269.534,A -85,B 0,C 180,E1 -19567.826,E2 -19567.826} C_VEL
LIN {X 0,Y 237.305,Z 265.952,A -85,B 0,C 180,E1 -19568.492,E2 -19568.492} C_VEL
LIN {X 0,Y 234.99,Z 258.368,A -85,B 0,C 180,E1 -19572.641,E2 -19572.641} C_VEL
LIN {X 0,Y 234.876,Z 257.742,A -85,B 0,C 180,E1 -19573.232,E2 -19573.232} C_VEL
LIN {X 0,Y 234.859,Z 257.728,A -85,B 0,C 180,E1 -19576.501,E2 -19576.501} C_VEL
LIN {X 0,Y 234.924,Z 257.715,A -85,B 0,C 180,E1 -19581.074,E2 -19581.074} C_VEL
LIN {X 0,Y 234.927,Z 257.714,A -85,B 0,C 180,E1 -19585.356,E2 -19585.356} C_VEL
LIN {X 0,Y 234.902,Z 257.717,A -85,B 0,C 180,E1 -19589.422,E2 -19589.422} C_VEL
LIN {X 0,Y 234.971,Z 257.71,A -85,B 0,C 180,E1 -19593.801,E2 -19593.801} C_VEL
LIN {X 0,Y 234.991,Z 257.712,A -85,B 0,C 180,E1 -19598.962,E2 -19598.962} C_VEL
LIN {X 0,Y 235.063,Z 257.697,A -85,B 0,C 180,E1 -19603.08,E2 -19603.08} C_VEL
LIN {X 0,Y 235.096,Z 257.693,A -85,B 0,C 180,E1 -19607.916,E2 -19607.916} C_VEL
LIN {X 0,Y 235.309,Z 257.659,A -85,B 0,C 180,E1 -19611.406,E2 -19611.406} C_VEL
LIN {X 0,Y 235.346,Z 257.665,A -85,B 0,C 180,E1 -19613.134,E2 -19613.134} C_VEL
LIN {X 0,Y 235.568,Z 257.641,A -85,B 0,C 180,E1 -19618.285,E2 -19618.285} C_VEL
LIN {X 0,Y 235.556,Z 257.631,A -85,B 0,C 180,E1 -19621.704,E2 -19621.704} C_VEL
LIN {X 0,Y 235.341,Z 257.665,A -85,B 0,C 180,E1 -19626.854,E2 -19626.854} C_VEL
LIN {X 0,Y 235.2,Z 257.679,A -85,B 0,C 180,E1 -19630.322,E2 -19630.322} C_VEL
LIN {X 0,Y 235.066,Z 257.707,A -85,B 0,C 180,E1 -19635.603,E2 -19635.603} C_VEL
LIN {X 0,Y 234.975,Z 257.715,A -85,B 0,C 180,E1 -19639.202,E2 -19639.202} C_VEL
LIN {X 0,Y 234.928,Z 257.716,A -85,B 0,C 180,E1 -19642.879,E2 -19642.879} C_VEL
LIN {X 0,Y 234.956,Z 257.794,A -85,B 0,C 180,E1 -19646.191,E2 -19646.191} C_VEL
LIN {X 0,Y 235.97,Z 261.316,A -85,B 0,C 180,E1 -19648.209,E2 -19648.209} C_VEL
LIN {X 0,Y 238.17,Z 265.246,A -85,B 0,C 180,E1 -19649.008,E2 -19649.008} C_VEL
LIN {X 0,Y 244.583,Z 275.812,A -85,B 0,C 180,E1 -19650.838,E2 -19650.838} C_VEL
LIN {X 0,Y 251.44,Z 288.901,A -85,B 0,C 180,E1 -19652.685,E2 -19652.685} C_VEL
LIN {X 0,Y 257.009,Z 301.629,A -85,B 0,C 180,E1 -19654.147,E2 -19654.147} C_VEL
LIN {X 0,Y 258.871,Z 306.687,A -85,B 0,C 180,E1 -19654.64,E2 -19654.64} C_VEL
LIN {X 0,Y 255.947,Z 368.94,A -85,B 0,C 180,E1 -19656.425,E2 -19656.425} C_VEL
LIN {X 0,Y 254.682,Z 381.887,A -85,B 0,C 180,E1 -19657.065,E2 -19657.065} C_VEL
LIN {X 0,Y 253,Z 394.78,A -85,B 0,C 180,E1 -19658.034,E2 -19658.034} C_VEL
LIN {X 0,Y 250.863,Z 406.975,A -85,B 0,C 180,E1 -19659.295,E2 -19659.295} C_VEL
LIN {X 0,Y 248.437,Z 418.293,A -85,B 0,C 180,E1 -19660.826,E2 -19660.826} C_VEL
LIN {X 0,Y 245.902,Z 428.418,A -85,B 0,C 180,E1 -19662.558,E2 -19662.558} C_VEL
LIN {X 0,Y 243.484,Z 437.102,A -85,B 0,C 180,E1 -19664.409,E2 -19664.409} C_VEL
LIN {X 0,Y 240.743,Z 446.209,A -85,B 0,C 180,E1 -19666.861,E2 -19666.861} C_VEL
LIN {X 0,Y 238.335,Z 454.036,A -85,B 0,C 180,E1 -19669.556,E2 -19669.556} C_VEL
LIN {X 0,Y 236.266,Z 460.432,A -85,B 0,C 180,E1 -19672.427,E2 -19672.427} C_VEL
LIN {X 0,Y 234.671,Z 465.28,A -85,B 0,C 180,E1 -19675.32,E2 -19675.32} C_VEL
LIN {X 0,Y 233.926,Z 467.782,A -85,B 0,C 180,E1 -19677.265,E2 -19677.265} C_VEL
LIN {X 0,Y 233.304,Z 469.658,A -85,B 0,C 180,E1 -19679.198,E2 -19679.198} C_VEL
LIN {X 0,Y 232.857,Z 471.042,A -85,B 0,C 180,E1 -19681.126,E2 -19681.126} C_VEL
LIN {X 0,Y 232.486,Z 471.901,A -85,B 0,C 180,E1 -19683.037,E2 -19683.037} C_VEL
LIN {X 0,Y 232.303,Z 472.285,A -85,B 0,C 180,E1 -19685.158,E2 -19685.158} C_VEL
LIN {X 0,Y 232.223,Z 472.188,A -85,B 0,C 180,E1 -19686.833,E2 -19686.833} C_VEL
LIN {X 0,Y 232.347,Z 471.163,A -85,B 0,C 180,E1 -19689.644,E2 -19689.644} C_VEL
LIN {X 0,Y 232.694,Z 469.094,A -85,B 0,C 180,E1 -19692.422,E2 -19692.422} C_VEL
LIN {X 0,Y 233.137,Z 466.561,A -85,B 0,C 180,E1 -19694.691,E2 -19694.691} C_VEL
LIN {X 0,Y 234.074,Z 461.696,A -85,B 0,C 180,E1 -19697.869,E2 -19697.869} C_VEL
LIN {X 0,Y 235.386,Z 455.241,A -85,B 0,C 180,E1 -19700.935,E2 -19700.935} C_VEL
LIN {X 0,Y 236.986,Z 447.94,A -85,B 0,C 180,E1 -19703.616,E2 -19703.616} C_VEL
LIN {X 0,Y 238.696,Z 440.216,A -85,B 0,C 180,E1 -19705.865,E2 -19705.865} C_VEL
LIN {X 0,Y 240.734,Z 430.549,A -85,B 0,C 180,E1 -19708.119,E2 -19708.119} C_VEL
LIN {X 0,Y 242.749,Z 420.436,A -85,B 0,C 180,E1 -19710.001,E2 -19710.001} C_VEL
LIN {X 0,Y 244.774,Z 409.186,A -85,B 0,C 180,E1 -19711.647,E2 -19711.647} C_VEL
LIN {X 0,Y 246.586,Z 396.557,A -85,B 0,C 180,E1 -19713.068,E2 -19713.068} C_VEL
LIN {X 0,Y 247.929,Z 384.66,A -85,B 0,C 180,E1 -19714.065,E2 -19714.065} C_VEL
LIN {X 0,Y 249.047,Z 371.599,A -85,B 0,C 180,E1 -19714.807,E2 -19714.807} C_VEL
LIN {X 0,Y 249.933,Z 353.459,A -85,B 0,C 180,E1 -19715.398,E2 -19715.398} C_VEL
LIN {X 0,Y 251.68,Z 302.868,A -85,B 0,C 180,E1 -19716.857,E2 -19716.857} C_VEL
LIN {X 0,Y 250.36,Z 295.924,A -85,B 0,C 180,E1 -19717.237,E2 -19717.237} C_VEL
LIN {X 0,Y 240.563,Z 271.291,A -85,B 0,C 180,E1 -19719.271,E2 -19719.271} C_VEL
LIN {X 0,Y 236.116,Z 261.591,A -85,B 0,C 180,E1 -19720.249,E2 -19720.249} C_VEL
LIN {X 0,Y 235.502,Z 259.391,A -85,B 0,C 180,E1 -19721.099,E2 -19721.099} C_VEL
LIN {X 0,Y 235.112,Z 257.711,A -85,B 0,C 180,E1 -19722.079,E2 -19722.079} C_VEL
LIN {X 0,Y 235.067,Z 257.698,A -85,B 0,C 180,E1 -19726.943,E2 -19726.943} C_VEL
LIN {X 0,Y 234.959,Z 257.72,A -85,B 0,C 180,E1 -19732.009,E2 -19732.009} C_VEL
LIN {X 0,Y 234.917,Z 257.724,A -85,B 0,C 180,E1 -19736.665,E2 -19736.665} C_VEL
LIN {X 0,Y 234.87,Z 257.719,A -85,B 0,C 180,E1 -19740.578,E2 -19740.578} C_VEL
LIN {X 0,Y 234.916,Z 257.719,A -85,B 0,C 180,E1 -19743.118,E2 -19743.118} C_VEL
LIN {X 0,Y 234.893,Z 257.713,A -85,B 0,C 180,E1 -19746.757,E2 -19746.757} C_VEL
LIN {X 0,Y 234.891,Z 257.727,A -85,B 0,C 180,E1 -19748.941,E2 -19748.941} C_VEL
LIN {X 0,Y 234.833,Z 257.711,A -85,B 0,C 180,E1 -19753.5,E2 -19753.5} C_VEL
LIN {X 0,Y 234.843,Z 257.732,A -85,B 0,C 180,E1 -19756.514,E2 -19756.514} C_VEL
LIN {X 0,Y 234.903,Z 257.69,A -85,B 0,C 180,E1 -19761.085,E2 -19761.085} C_VEL
LIN {X 0,Y 234.909,Z 257.723,A -85,B 0,C 180,E1 -19765.367,E2 -19765.367} C_VEL
LIN {X 0,Y 234.883,Z 257.701,A -85,B 0,C 180,E1 -19769.433,E2 -19769.433} C_VEL
LIN {X 0,Y 234.931,Z 257.701,A -85,B 0,C 180,E1 -19773.828,E2 -19773.828} C_VEL
LIN {X 0,Y 234.979,Z 257.704,A -85,B 0,C 180,E1 -19778.974,E2 -19778.974} C_VEL
LIN {X 0,Y 235.053,Z 257.659,A -85,B 0,C 180,E1 -19783.099,E2 -19783.099} C_VEL
LIN {X 0,Y 235.107,Z 257.7,A -85,B 0,C 180,E1 -19787.928,E2 -19787.928} C_VEL
LIN {X 0,Y 235.311,Z 257.651,A -85,B 0,C 180,E1 -19791.418,E2 -19791.418} C_VEL
LIN {X 0,Y 235.348,Z 257.626,A -85,B 0,C 180,E1 -19793.146,E2 -19793.146} C_VEL
LIN {X 0,Y 235.578,Z 257.633,A -85,B 0,C 180,E1 -19798.296,E2 -19798.296} C_VEL
LIN {X 0,Y 235.58,Z 257.63,A -85,B 0,C 180,E1 -19801.715,E2 -19801.715} C_VEL
LIN {X 0,Y 235.365,Z 257.636,A -85,B 0,C 180,E1 -19806.865,E2 -19806.865} C_VEL
LIN {X 0,Y 235.222,Z 257.685,A -85,B 0,C 180,E1 -19810.333,E2 -19810.333} C_VEL
LIN {X 0,Y 235.09,Z 257.667,A -85,B 0,C 180,E1 -19815.613,E2 -19815.613} C_VEL
LIN {X 0,Y 235,Z 257.713,A -85,B 0,C 180,E1 -19819.212,E2 -19819.212} C_VEL
LIN {X 0,Y 234.963,Z 257.696,A -85,B 0,C 180,E1 -19822.632,E2 -19822.632} C_VEL
LIN {X 0,Y 234.263,Z 257.779,A -85,B 0,C 180,E1 -19824.063,E2 -19824.063} C_VEL
LIN {X 0,Y 231.386,Z 258.156,A -85,B 0,C 180,E1 -19826.397,E2 -19826.397} C_VEL
LIN {X 0,Y 228.972,Z 258.463,A -85,B 0,C 180,E1 -19828.301,E2 -19828.301} C_VEL
LIN {X 0,Y 227.958,Z 258.579,A -85,B 0,C 180,E1 -19829.778,E2 -19829.778} C_VEL
LIN {X 0,Y 227.887,Z 258.582,A -85,B 0,C 180,E1 -19830.279,E2 -19830.279} C_VEL
LIN {X 0,Y 227.89,Z 258.596,A -85,B 0,C 180,E1 -19833.724,E2 -19833.724} C_VEL
LIN {X 0,Y 227.855,Z 258.589,A -85,B 0,C 180,E1 -19838.095,E2 -19838.095} C_VEL
LIN {X 0,Y 227.8,Z 258.596,A -85,B 0,C 180,E1 -19842.751,E2 -19842.751} C_VEL
LIN {X 0,Y 227.807,Z 258.604,A -85,B 0,C 180,E1 -19847.255,E2 -19847.255} C_VEL
LIN {X 0,Y 227.96,Z 258.72,A -85,B 0,C 180,E1 -19852.109,E2 -19852.109} C_VEL
LIN {X 0,Y 229.857,Z 266.918,A -85,B 0,C 180,E1 -19855.885,E2 -19855.885} C_VEL
LIN {X 0,Y 237.988,Z 286.112,A -85,B 0,C 180,E1 -19857.751,E2 -19857.751} C_VEL
LIN {X 0,Y 242.535,Z 298.528,A -85,B 0,C 180,E1 -19858.753,E2 -19858.753} C_VEL
LIN {X 0,Y 245.052,Z 315.433,A -85,B 0,C 180,E1 -19859.632,E2 -19859.632} C_VEL
LIN {X 0,Y 242.723,Z 374.697,A -85,B 0,C 180,E1 -19861.401,E2 -19861.401} C_VEL
LIN {X 0,Y 241.634,Z 387.82,A -85,B 0,C 180,E1 -19862.088,E2 -19862.088} C_VEL
LIN {X 0,Y 240.008,Z 401.073,A -85,B 0,C 180,E1 -19863.124,E2 -19863.124} C_VEL
LIN {X 0,Y 238.171,Z 413.042,A -85,B 0,C 180,E1 -19864.432,E2 -19864.432} C_VEL
LIN {X 0,Y 236.104,Z 424.531,A -85,B 0,C 180,E1 -19866.072,E2 -19866.072} C_VEL
LIN {X 0,Y 233.938,Z 434.885,A -85,B 0,C 180,E1 -19867.942,E2 -19867.942} C_VEL
LIN {X 0,Y 232.113,Z 443.975,A -85,B 0,C 180,E1 -19870.023,E2 -19870.023} C_VEL
LIN {X 0,Y 230.266,Z 451.84,A -85,B 0,C 180,E1 -19872.228,E2 -19872.228} C_VEL
LIN {X 0,Y 228.568,Z 459.337,A -85,B 0,C 180,E1 -19874.848,E2 -19874.848} C_VEL
LIN {X 0,Y 227.291,Z 465.346,A -85,B 0,C 180,E1 -19877.498,E2 -19877.498} C_VEL
LIN {X 0,Y 226.391,Z 470.079,A -85,B 0,C 180,E1 -19880.168,E2 -19880.168} C_VEL
LIN {X 0,Y 225.843,Z 473.678,A -85,B 0,C 180,E1 -19882.848,E2 -19882.848} C_VEL
LIN {X 0,Y 225.597,Z 476.25,A -85,B 0,C 180,E1 -19885.533,E2 -19885.533} C_VEL
LIN {X 0,Y 225.576,Z 477.863,A -85,B 0,C 180,E1 -19888.213,E2 -19888.213} C_VEL
LIN {X 0,Y 225.644,Z 478.443,A -85,B 0,C 180,E1 -19889.999,E2 -19889.999} C_VEL
LIN {X 0,Y 225.577,Z 478.61,A -85,B 0,C 180,E1 -19891.784,E2 -19891.784} C_VEL
LIN {X 0,Y 225.666,Z 477.708,A -85,B 0,C 180,E1 -19895.359,E2 -19895.359} C_VEL
LIN {X 0,Y 225.932,Z 476.68,A -85,B 0,C 180,E1 -19897.146,E2 -19897.146} C_VEL
LIN {X 0,Y 226.268,Z 475.239,A -85,B 0,C 180,E1 -19898.933,E2 -19898.933} C_VEL
LIN {X 0,Y 227.092,Z 472.265,A -85,B 0,C 180,E1 -19901.603,E2 -19901.603} C_VEL
LIN {X 0,Y 228.322,Z 468.262,A -85,B 0,C 180,E1 -19904.254,E2 -19904.254} C_VEL
LIN {X 0,Y 230.441,Z 462.122,A -85,B 0,C 180,E1 -19907.297,E2 -19907.297} C_VEL
LIN {X 0,Y 232.727,Z 455.445,A -85,B 0,C 180,E1 -19909.859,E2 -19909.859} C_VEL
LIN {X 0,Y 235.051,Z 447.786,A -85,B 0,C 180,E1 -19912.221,E2 -19912.221} C_VEL
LIN {X 0,Y 237.751,Z 438.734,A -85,B 0,C 180,E1 -19914.445,E2 -19914.445} C_VEL
LIN {X 0,Y 240.736,Z 428.306,A -85,B 0,C 180,E1 -19916.435,E2 -19916.435} C_VEL
LIN {X 0,Y 243.248,Z 418.027,A -85,B 0,C 180,E1 -19918,E2 -19918} C_VEL
LIN {X 0,Y 245.658,Z 406.795,A -85,B 0,C 180,E1 -19919.334,E2 -19919.334} C_VEL
LIN {X 0,Y 247.778,Z 394.12,A -85,B 0,C 180,E1 -19920.463,E2 -19920.463} C_VEL
LIN {X 0,Y 249.322,Z 381.919,A -85,B 0,C 180,E1 -19921.231,E2 -19921.231} C_VEL
LIN {X 0,Y 250.475,Z 368.477,A -85,B 0,C 180,E1 -19921.758,E2 -19921.758} C_VEL
LIN {X 0,Y 252.709,Z 317.192,A -85,B 0,C 180,E1 -19923.267,E2 -19923.267} C_VEL
LIN {X 0,Y 251.064,Z 307.122,A -85,B 0,C 180,E1 -19923.937,E2 -19923.937} C_VEL
LIN {X 0,Y 245.47,Z 294.194,A -85,B 0,C 180,E1 -19925.486,E2 -19925.486} C_VEL
LIN {X 0,Y 239.723,Z 282.791,A -85,B 0,C 180,E1 -19927.143,E2 -19927.143} C_VEL
LIN {X 0,Y 234.922,Z 274.267,A -85,B 0,C 180,E1 -19928.588,E2 -19928.588} C_VEL
LIN {X 0,Y 232.129,Z 269.665,A -85,B 0,C 180,E1 -19929.457,E2 -19929.457} C_VEL
LIN {X 0,Y 229.928,Z 265.761,A -85,B 0,C 180,E1 -19930.302,E2 -19930.302} C_VEL
LIN {X 0,Y 227.881,Z 258.906,A -85,B 0,C 180,E1 -19934.347,E2 -19934.347} C_VEL
LIN {X 0,Y 227.818,Z 258.604,A -85,B 0,C 180,E1 -19935.194,E2 -19935.194} C_VEL
LIN {X 0,Y 227.806,Z 258.608,A -85,B 0,C 180,E1 -19939.613,E2 -19939.613} C_VEL
LIN {X 0,Y 227.869,Z 258.595,A -85,B 0,C 180,E1 -19944.12,E2 -19944.12} C_VEL
LIN {X 0,Y 227.859,Z 258.592,A -85,B 0,C 180,E1 -19948.37,E2 -19948.37} C_VEL
LIN {X 0,Y 227.857,Z 258.591,A -85,B 0,C 180,E1 -19952.436,E2 -19952.436} C_VEL
LIN {X 0,Y 227.895,Z 258.587,A -85,B 0,C 180,E1 -19956.36,E2 -19956.36} C_VEL
LIN {X 0,Y 227.926,Z 258.59,A -85,B 0,C 180,E1 -19960.167,E2 -19960.167} C_VEL
LIN {X 0,Y 228.028,Z 258.581,A -85,B 0,C 180,E1 -19963.89,E2 -19963.89} C_VEL
LIN {X 0,Y 228.054,Z 258.566,A -85,B 0,C 180,E1 -19967.536,E2 -19967.536} C_VEL
LIN {X 0,Y 228.251,Z 258.539,A -85,B 0,C 180,E1 -19971.138,E2 -19971.138} C_VEL
LIN {X 0,Y 228.299,Z 258.541,A -85,B 0,C 180,E1 -19972.921,E2 -19972.921} C_VEL
LIN {X 0,Y 228.526,Z 258.517,A -85,B 0,C 180,E1 -19978.232,E2 -19978.232} C_VEL
LIN {X 0,Y 228.49,Z 258.511,A -85,B 0,C 180,E1 -19981.757,E2 -19981.757} C_VEL
LIN {X 0,Y 228.293,Z 258.545,A -85,B 0,C 180,E1 -19987.067,E2 -19987.067} C_VEL
LIN {X 0,Y 228.13,Z 258.561,A -85,B 0,C 180,E1 -19990.645,E2 -19990.645} C_VEL
LIN {X 0,Y 228.024,Z 258.575,A -85,B 0,C 180,E1 -19994.268,E2 -19994.268} C_VEL
LIN {X 0,Y 227.94,Z 258.588,A -85,B 0,C 180,E1 -19997.951,E2 -19997.951} C_VEL
LIN {X 0,Y 227.92,Z 258.591,A -85,B 0,C 180,E1 -20002.327,E2 -20002.327} C_VEL
LIN {X 0,Y 227.938,Z 258.799,A -85,B 0,C 180,E1 -20004.833,E2 -20004.833} C_VEL
LIN {X 0,Y 228.833,Z 261.737,A -85,B 0,C 180,E1 -20006.53,E2 -20006.53} C_VEL
LIN {X 0,Y 232.946,Z 268.476,A -85,B 0,C 180,E1 -20007.934,E2 -20007.934} C_VEL
LIN {X 0,Y 239.944,Z 280,A -85,B 0,C 180,E1 -20010.033,E2 -20010.033} C_VEL
LIN {X 0,Y 246.764,Z 293.232,A -85,B 0,C 180,E1 -20011.972,E2 -20011.972} C_VEL
LIN {X 0,Y 252.884,Z 307.545,A -85,B 0,C 180,E1 -20013.647,E2 -20013.647} C_VEL
LIN {X 0,Y 253.135,Z 309.076,A -85,B 0,C 180,E1 -20013.749,E2 -20013.749} C_VEL
LIN {X 0,Y 250.151,Z 369.032,A -85,B 0,C 180,E1 -20015.501,E2 -20015.501} C_VEL
LIN {X 0,Y 248.878,Z 381.587,A -85,B 0,C 180,E1 -20016.127,E2 -20016.127} C_VEL
LIN {X 0,Y 247.208,Z 393.985,A -85,B 0,C 180,E1 -20017.062,E2 -20017.062} C_VEL
LIN {X 0,Y 245.086,Z 405.925,A -85,B 0,C 180,E1 -20018.282,E2 -20018.282} C_VEL
LIN {X 0,Y 242.578,Z 417.321,A -85,B 0,C 180,E1 -20019.819,E2 -20019.819} C_VEL
LIN {X 0,Y 239.804,Z 427.963,A -85,B 0,C 180,E1 -20021.643,E2 -20021.643} C_VEL
LIN {X 0,Y 237.305,Z 436.549,A -85,B 0,C 180,E1 -20023.485,E2 -20023.485} C_VEL
LIN {X 0,Y 234.677,Z 445,A -85,B 0,C 180,E1 -20025.74,E2 -20025.74} C_VEL
LIN {X 0,Y 232.256,Z 452.467,A -85,B 0,C 180,E1 -20028.265,E2 -20028.265} C_VEL
LIN {X 0,Y 229.884,Z 459.244,A -85,B 0,C 180,E1 -20031.193,E2 -20031.193} C_VEL
LIN {X 0,Y 228.115,Z 464.444,A -85,B 0,C 180,E1 -20034.173,E2 -20034.173} C_VEL
LIN {X 0,Y 227.021,Z 467.704,A -85,B 0,C 180,E1 -20036.691,E2 -20036.691} C_VEL
LIN {X 0,Y 226.492,Z 469.199,A -85,B 0,C 180,E1 -20038.165,E2 -20038.165} C_VEL
LIN {X 0,Y 225.851,Z 470.996,A -85,B 0,C 180,E1 -20040.594,E2 -20040.594} C_VEL
LIN {X 0,Y 225.253,Z 472.312,A -85,B 0,C 180,E1 -20044.102,E2 -20044.102} C_VEL
LIN {X 0,Y 225.151,Z 472.351,A -85,B 0,C 180,E1 -20046.061,E2 -20046.061} C_VEL
LIN {X 0,Y 225.23,Z 471.368,A -85,B 0,C 180,E1 -20049.386,E2 -20049.386} C_VEL
LIN {X 0,Y 225.473,Z 469.723,A -85,B 0,C 180,E1 -20051.84,E2 -20051.84} C_VEL
LIN {X 0,Y 226.007,Z 466.988,A -85,B 0,C 180,E1 -20054.547,E2 -20054.547} C_VEL
LIN {X 0,Y 226.804,Z 462.834,A -85,B 0,C 180,E1 -20057.474,E2 -20057.474} C_VEL
LIN {X 0,Y 228.022,Z 457.172,A -85,B 0,C 180,E1 -20060.454,E2 -20060.454} C_VEL
LIN {X 0,Y 229.678,Z 449.757,A -85,B 0,C 180,E1 -20063.412,E2 -20063.412} C_VEL
LIN {X 0,Y 231.658,Z 441.188,A -85,B 0,C 180,E1 -20066.087,E2 -20066.087} C_VEL
LIN {X 0,Y 233.604,Z 432.34,A -85,B 0,C 180,E1 -20068.277,E2 -20068.277} C_VEL
LIN {X 0,Y 235.916,Z 421.342,A -85,B 0,C 180,E1 -20070.428,E2 -20070.428} C_VEL
LIN {X 0,Y 237.998,Z 410.349,A -85,B 0,C 180,E1 -20072.117,E2 -20072.117} C_VEL
LIN {X 0,Y 239.853,Z 398.052,A -85,B 0,C 180,E1 -20073.571,E2 -20073.571} C_VEL
LIN {X 0,Y 241.398,Z 385.201,A -85,B 0,C 180,E1 -20074.698,E2 -20074.698} C_VEL
LIN {X 0,Y 242.54,Z 372.728,A -85,B 0,C 180,E1 -20075.445,E2 -20075.445} C_VEL
LIN {X 0,Y 243.356,Z 356.794,A -85,B 0,C 180,E1 -20076.006,E2 -20076.006} C_VEL
LIN {X 0,Y 245.342,Z 303.904,A -85,B 0,C 180,E1 -20077.558,E2 -20077.558} C_VEL
LIN {X 0,Y 244.333,Z 298.534,A -85,B 0,C 180,E1 -20077.861,E2 -20077.861} C_VEL
LIN {X 0,Y 234.847,Z 274.582,A -85,B 0,C 180,E1 -20079.901,E2 -20079.901} C_VEL
LIN {X 0,Y 228.79,Z 261.604,A -85,B 0,C 180,E1 -20081.275,E2 -20081.275} C_VEL
LIN {X 0,Y 228.092,Z 258.922,A -85,B 0,C 180,E1 -20082.457,E2 -20082.457} C_VEL
LIN {X 0,Y 228.03,Z 258.567,A -85,B 0,C 180,E1 -20082.913,E2 -20082.913} C_VEL
LIN {X 0,Y 228.005,Z 258.578,A -85,B 0,C 180,E1 -20087.176,E2 -20087.176} C_VEL
LIN {X 0,Y 227.892,Z 258.598,A -85,B 0,C 180,E1 -20092.326,E2 -20092.326} C_VEL
LIN {X 0,Y 227.895,Z 258.599,A -85,B 0,C 180,E1 -20096.596,E2 -20096.596} C_VEL
LIN {X 0,Y 227.845,Z 258.59,A -85,B 0,C 180,E1 -20100.284,E2 -20100.284} C_VEL
LIN {X 0,Y 227.849,Z 258.592,A -85,B 0,C 180,E1 -20103.727,E2 -20103.727} C_VEL
LIN {X 0,Y 227.819,Z 258.606,A -85,B 0,C 180,E1 -20108.098,E2 -20108.098} C_VEL
LIN {X 0,Y 227.765,Z 258.587,A -85,B 0,C 180,E1 -20112.755,E2 -20112.755} C_VEL
LIN {X 0,Y 227.773,Z 258.611,A -85,B 0,C 180,E1 -20117.259,E2 -20117.259} C_VEL
LIN {X 0,Y 227.825,Z 258.573,A -85,B 0,C 180,E1 -20121.914,E2 -20121.914} C_VEL
LIN {X 0,Y 227.866,Z 258.6,A -85,B 0,C 180,E1 -20126.385,E2 -20126.385} C_VEL
LIN {X 0,Y 227.86,Z 258.563,A -85,B 0,C 180,E1 -20130.437,E2 -20130.437} C_VEL
LIN {X 0,Y 227.863,Z 258.59,A -85,B 0,C 180,E1 -20134.426,E2 -20134.426} C_VEL
LIN {X 0,Y 227.939,Z 258.586,A -85,B 0,C 180,E1 -20138.292,E2 -20138.292} C_VEL
LIN {X 0,Y 228.02,Z 258.541,A -85,B 0,C 180,E1 -20143.902,E2 -20143.902} C_VEL
LIN {X 0,Y 228.063,Z 258.574,A -85,B 0,C 180,E1 -20147.549,E2 -20147.549} C_VEL
LIN {X 0,Y 228.253,Z 258.533,A -85,B 0,C 180,E1 -20151.15,E2 -20151.15} C_VEL
LIN {X 0,Y 228.3,Z 258.505,A -85,B 0,C 180,E1 -20152.933,E2 -20152.933} C_VEL
LIN {X 0,Y 228.537,Z 258.51,A -85,B 0,C 180,E1 -20158.244,E2 -20158.244} C_VEL
LIN {X 0,Y 228.538,Z 258.506,A -85,B 0,C 180,E1 -20161.768,E2 -20161.768} C_VEL
LIN {X 0,Y 228.317,Z 258.516,A -85,B 0,C 180,E1 -20167.078,E2 -20167.078} C_VEL
LIN {X 0,Y 228.153,Z 258.566,A -85,B 0,C 180,E1 -20170.657,E2 -20170.657} C_VEL
LIN {X 0,Y 228.055,Z 258.547,A -85,B 0,C 180,E1 -20174.278,E2 -20174.278} C_VEL
LIN {X 0,Y 227.965,Z 258.58,A -85,B 0,C 180,E1 -20177.962,E2 -20177.962} C_VEL
LIN {X 0,Y 227.915,Z 258.573,A -85,B 0,C 180,E1 -20182.613,E2 -20182.613} C_VEL
LIN {X 0,Y 227.935,Z 258.586,A -85,B 0,C 180,E1 -20186.596,E2 -20186.596} C_VEL
LIN {X 0,Y 227.887,Z 258.582,A -85,B 0,C 180,E1 -20190.279,E2 -20190.279} C_VEL
LIN {X 0,Y 227.243,Z 258.663,A -85,B 0,C 180,E1 -20191.754,E2 -20191.754} C_VEL
LIN {X 0,Y 224.386,Z 259.035,A -85,B 0,C 180,E1 -20194.159,E2 -20194.159} C_VEL
LIN {X 0,Y 221.93,Z 259.332,A -85,B 0,C 180,E1 -20196.121,E2 -20196.121} C_VEL
LIN {X 0,Y 220.861,Z 259.458,A -85,B 0,C 180,E1 -20197.646,E2 -20197.646} C_VEL
LIN {X 0,Y 220.767,Z 259.47,A -85,B 0,C 180,E1 -20198.163,E2 -20198.163} C_VEL
LIN {X 0,Y 220.763,Z 259.473,A -85,B 0,C 180,E1 -20201.961,E2 -20201.961} C_VEL
LIN {X 0,Y 220.771,Z 259.481,A -85,B 0,C 180,E1 -20205.544,E2 -20205.544} C_VEL
LIN {X 0,Y 220.798,Z 259.481,A -85,B 0,C 180,E1 -20210.46,E2 -20210.46} C_VEL
LIN {X 0,Y 220.893,Z 259.693,A -85,B 0,C 180,E1 -20211.405,E2 -20211.405} C_VEL
LIN {X 0,Y 222.581,Z 266.798,A -85,B 0,C 180,E1 -20214.806,E2 -20214.806} C_VEL
LIN {X 0,Y 227.836,Z 278.815,A -85,B 0,C 180,E1 -20216.104,E2 -20216.104} C_VEL
LIN {X 0,Y 233.818,Z 293.274,A -85,B 0,C 180,E1 -20217.458,E2 -20217.458} C_VEL
LIN {X 0,Y 236.427,Z 300.812,A -85,B 0,C 180,E1 -20218.068,E2 -20218.068} C_VEL
LIN {X 0,Y 238.665,Z 317.063,A -85,B 0,C 180,E1 -20218.919,E2 -20218.919} C_VEL
LIN {X 0,Y 236.326,Z 374.482,A -85,B 0,C 180,E1 -20220.674,E2 -20220.674} C_VEL
LIN {X 0,Y 235.171,Z 387.633,A -85,B 0,C 180,E1 -20221.373,E2 -20221.373} C_VEL
LIN {X 0,Y 233.528,Z 400.918,A -85,B 0,C 180,E1 -20222.437,E2 -20222.437} C_VEL
LIN {X 0,Y 231.77,Z 412.112,A -85,B 0,C 180,E1 -20223.673,E2 -20223.673} C_VEL
LIN {X 0,Y 229.583,Z 423.751,A -85,B 0,C 180,E1 -20225.348,E2 -20225.348} C_VEL
LIN {X 0,Y 227.368,Z 434.235,A -85,B 0,C 180,E1 -20227.269,E2 -20227.269} C_VEL
LIN {X 0,Y 225.229,Z 444.234,A -85,B 0,C 180,E1 -20229.612,E2 -20229.612} C_VEL
LIN {X 0,Y 223.138,Z 452.761,A -85,B 0,C 180,E1 -20232.115,E2 -20232.115} C_VEL
LIN {X 0,Y 221.412,Z 460.079,A -85,B 0,C 180,E1 -20234.818,E2 -20234.818} C_VEL
LIN {X 0,Y 220.307,Z 465.015,A -85,B 0,C 180,E1 -20237.095,E2 -20237.095} C_VEL
LIN {X 0,Y 219.372,Z 469.799,A -85,B 0,C 180,E1 -20239.85,E2 -20239.85} C_VEL
LIN {X 0,Y 218.782,Z 473.445,A -85,B 0,C 180,E1 -20242.616,E2 -20242.616} C_VEL
LIN {X 0,Y 218.497,Z 476.315,A -85,B 0,C 180,E1 -20245.709,E2 -20245.709} C_VEL
LIN {X 0,Y 218.478,Z 477.714,A -85,B 0,C 180,E1 -20248.155,E2 -20248.155} C_VEL
LIN {X 0,Y 218.543,Z 478.314,A -85,B 0,C 180,E1 -20249.998,E2 -20249.998} C_VEL
LIN {X 0,Y 218.48,Z 478.515,A -85,B 0,C 180,E1 -20251.842,E2 -20251.842} C_VEL
LIN {X 0,Y 218.591,Z 477.663,A -85,B 0,C 180,E1 -20255.533,E2 -20255.533} C_VEL
LIN {X 0,Y 218.868,Z 476.657,A -85,B 0,C 180,E1 -20257.378,E2 -20257.378} C_VEL
LIN {X 0,Y 219.233,Z 475.255,A -85,B 0,C 180,E1 -20259.222,E2 -20259.222} C_VEL
LIN {X 0,Y 220.132,Z 472.321,A -85,B 0,C 180,E1 -20261.975,E2 -20261.975} C_VEL
LIN {X 0,Y 221.422,Z 468.364,A -85,B 0,C 180,E1 -20264.708,E2 -20264.708} C_VEL
LIN {X 0,Y 223.339,Z 463.287,A -85,B 0,C 180,E1 -20267.393,E2 -20267.393} C_VEL
LIN {X 0,Y 225.605,Z 456.917,A -85,B 0,C 180,E1 -20270.038,E2 -20270.038} C_VEL
LIN {X 0,Y 228.124,Z 449.277,A -85,B 0,C 180,E1 -20272.552,E2 -20272.552} C_VEL
LIN {X 0,Y 230.769,Z 440.921,A -85,B 0,C 180,E1 -20274.754,E2 -20274.754} C_VEL
LIN {X 0,Y 233.775,Z 431.122,A -85,B 0,C 180,E1 -20276.803,E2 -20276.803} C_VEL
LIN {X 0,Y 236.694,Z 420.179,A -85,B 0,C 180,E1 -20278.604,E2 -20278.604} C_VEL
LIN {X 0,Y 239.553,Z 407.756,A -85,B 0,C 180,E1 -20280.158,E2 -20280.158} C_VEL
LIN {X 0,Y 241.75,Z 395.585,A -85,B 0,C 180,E1 -20281.307,E2 -20281.307} C_VEL
LIN {X 0,Y 243.485,Z 382.815,A -85,B 0,C 180,E1 -20282.151,E2 -20282.151} C_VEL
LIN {X 0,Y 244.616,Z 370.937,A -85,B 0,C 180,E1 -20282.654,E2 -20282.654} C_VEL
LIN {X 0,Y 247.072,Z 318.485,A -85,B 0,C 180,E1 -20284.233,E2 -20284.233} C_VEL
LIN {X 0,Y 245.742,Z 310.065,A -85,B 0,C 180,E1 -20284.81,E2 -20284.81} C_VEL
LIN {X 0,Y 239.814,Z 296.23,A -85,B 0,C 180,E1 -20286.559,E2 -20286.559} C_VEL
LIN {X 0,Y 233.773,Z 284.318,A -85,B 0,C 180,E1 -20288.409,E2 -20288.409} C_VEL
LIN {X 0,Y 228.187,Z 274.748,A -85,B 0,C 180,E1 -20290.208,E2 -20290.208} C_VEL
LIN {X 0,Y 224.914,Z 269.663,A -85,B 0,C 180,E1 -20291.332,E2 -20291.332} C_VEL
LIN {X 0,Y 222.618,Z 265.625,A -85,B 0,C 180,E1 -20292.298,E2 -20292.298} C_VEL
LIN {X 0,Y 220.754,Z 259.623,A -85,B 0,C 180,E1 -20296.174,E2 -20296.174} C_VEL
LIN {X 0,Y 220.787,Z 259.48,A -85,B 0,C 180,E1 -20300.452,E2 -20300.452} C_VEL
LIN {X 0,Y 220.831,Z 259.476,A -85,B 0,C 180,E1 -20302.788,E2 -20302.788} C_VEL
LIN {X 0,Y 220.816,Z 259.477,A -85,B 0,C 180,E1 -20307.238,E2 -20307.238} C_VEL
LIN {X 0,Y 220.807,Z 259.475,A -85,B 0,C 180,E1 -20311.476,E2 -20311.476} C_VEL
LIN {X 0,Y 220.849,Z 259.472,A -85,B 0,C 180,E1 -20315.557,E2 -20315.557} C_VEL
LIN {X 0,Y 220.88,Z 259.472,A -85,B 0,C 180,E1 -20319.507,E2 -20319.507} C_VEL
LIN {X 0,Y 220.99,Z 259.452,A -85,B 0,C 180,E1 -20323.362,E2 -20323.362} C_VEL
LIN {X 0,Y 221.06,Z 259.449,A -85,B 0,C 180,E1 -20328.997,E2 -20328.997} C_VEL
LIN {X 0,Y 221.236,Z 259.417,A -85,B 0,C 180,E1 -20332.694,E2 -20332.694} C_VEL
LIN {X 0,Y 221.459,Z 259.396,A -85,B 0,C 180,E1 -20338.175,E2 -20338.175} C_VEL
LIN {X 0,Y 221.531,Z 259.381,A -85,B 0,C 180,E1 -20339.994,E2 -20339.994} C_VEL
LIN {X 0,Y 221.427,Z 259.391,A -85,B 0,C 180,E1 -20341.813,E2 -20341.813} C_VEL
LIN {X 0,Y 221.231,Z 259.426,A -85,B 0,C 180,E1 -20347.294,E2 -20347.294} C_VEL
LIN {X 0,Y 221.05,Z 259.446,A -85,B 0,C 180,E1 -20350.991,E2 -20350.991} C_VEL
LIN {X 0,Y 220.965,Z 259.455,A -85,B 0,C 180,E1 -20356.627,E2 -20356.627} C_VEL
LIN {X 0,Y 220.863,Z 259.468,A -85,B 0,C 180,E1 -20360.482,E2 -20360.482} C_VEL
LIN {X 0,Y 220.862,Z 259.612,A -85,B 0,C 180,E1 -20363.099,E2 -20363.099} C_VEL
LIN {X 0,Y 221.593,Z 261.884,A -85,B 0,C 180,E1 -20364.529,E2 -20364.529} C_VEL
LIN {X 0,Y 224.586,Z 266.451,A -85,B 0,C 180,E1 -20365.664,E2 -20365.664} C_VEL
LIN {X 0,Y 228.981,Z 273.546,A -85,B 0,C 180,E1 -20367.183,E2 -20367.183} C_VEL
LIN {X 0,Y 235.743,Z 284.965,A -85,B 0,C 180,E1 -20369.318,E2 -20369.318} C_VEL
LIN {X 0,Y 242.18,Z 297.701,A -85,B 0,C 180,E1 -20371.238,E2 -20371.238} C_VEL
LIN {X 0,Y 247.471,Z 310.277,A -85,B 0,C 180,E1 -20372.767,E2 -20372.767} C_VEL
LIN {X 0,Y 244.408,Z 369.721,A -85,B 0,C 180,E1 -20374.552,E2 -20374.552} C_VEL
LIN {X 0,Y 243.032,Z 382.5,A -85,B 0,C 180,E1 -20375.214,E2 -20375.214} C_VEL
LIN {X 0,Y 241.185,Z 395.319,A -85,B 0,C 180,E1 -20376.219,E2 -20376.219} C_VEL
LIN {X 0,Y 239,Z 406.772,A -85,B 0,C 180,E1 -20377.446,E2 -20377.446} C_VEL
LIN {X 0,Y 236.422,Z 417.852,A -85,B 0,C 180,E1 -20378.986,E2 -20378.986} C_VEL
LIN {X 0,Y 233.494,Z 428.516,A -85,B 0,C 180,E1 -20380.868,E2 -20380.868} C_VEL
LIN {X 0,Y 230.585,Z 437.958,A -85,B 0,C 180,E1 -20382.991,E2 -20382.991} C_VEL
LIN {X 0,Y 227.616,Z 446.781,A -85,B 0,C 180,E1 -20385.509,E2 -20385.509} C_VEL
LIN {X 0,Y 225.406,Z 453.282,A -85,B 0,C 180,E1 -20387.846,E2 -20387.846} C_VEL
LIN {X 0,Y 222.928,Z 460.021,A -85,B 0,C 180,E1 -20390.914,E2 -20390.914} C_VEL
LIN {X 0,Y 221.08,Z 465.014,A -85,B 0,C 180,E1 -20393.98,E2 -20393.98} C_VEL
LIN {X 0,Y 219.758,Z 468.644,A -85,B 0,C 180,E1 -20397.068,E2 -20397.068} C_VEL
LIN {X 0,Y 218.87,Z 470.997,A -85,B 0,C 180,E1 -20400.093,E2 -20400.093} C_VEL
LIN {X 0,Y 218.266,Z 472.27,A -85,B 0,C 180,E1 -20403.208,E2 -20403.208} C_VEL
LIN {X 0,Y 218.092,Z 472.51,A -85,B 0,C 180,E1 -20405.235,E2 -20405.235} C_VEL
LIN {X 0,Y 218.008,Z 472.231,A -85,B 0,C 180,E1 -20407.243,E2 -20407.243} C_VEL
LIN {X 0,Y 218.116,Z 471.511,A -85,B 0,C 180,E1 -20409.243,E2 -20409.243} C_VEL
LIN {X 0,Y 218.286,Z 470.345,A -85,B 0,C 180,E1 -20411.22,E2 -20411.22} C_VEL
LIN {X 0,Y 218.863,Z 467.395,A -85,B 0,C 180,E1 -20414.408,E2 -20414.408} C_VEL
LIN {X 0,Y 219.557,Z 463.935,A -85,B 0,C 180,E1 -20417.054,E2 -20417.054} C_VEL
LIN {X 0,Y 220.895,Z 457.899,A -85,B 0,C 180,E1 -20420.454,E2 -20420.454} C_VEL
LIN {X 0,Y 222.387,Z 451.537,A -85,B 0,C 180,E1 -20423.195,E2 -20423.195} C_VEL
LIN {X 0,Y 224.331,Z 443.34,A -85,B 0,C 180,E1 -20425.959,E2 -20425.959} C_VEL
LIN {X 0,Y 226.277,Z 434.942,A -85,B 0,C 180,E1 -20428.222,E2 -20428.222} C_VEL
LIN {X 0,Y 228.624,Z 424.622,A -85,B 0,C 180,E1 -20430.442,E2 -20430.442} C_VEL
LIN {X 0,Y 230.676,Z 414.36,A -85,B 0,C 180,E1 -20432.184,E2 -20432.184} C_VEL
LIN {X 0,Y 232.666,Z 402.857,A -85,B 0,C 180,E1 -20433.717,E2 -20433.717} C_VEL
LIN {X 0,Y 234.268,Z 390.837,A -85,B 0,C 180,E1 -20434.951,E2 -20434.951} C_VEL
LIN {X 0,Y 235.661,Z 377.958,A -85,B 0,C 180,E1 -20435.885,E2 -20435.885} C_VEL
LIN {X 0,Y 236.674,Z 364.309,A -85,B 0,C 180,E1 -20436.502,E2 -20436.502} C_VEL
LIN {X 0,Y 238.993,Z 304.515,A -85,B 0,C 180,E1 -20438.31,E2 -20438.31} C_VEL
LIN {X 0,Y 238.171,Z 300.806,A -85,B 0,C 180,E1 -20438.542,E2 -20438.542} C_VEL
LIN {X 0,Y 229.078,Z 277.715,A -85,B 0,C 180,E1 -20440.579,E2 -20440.579} C_VEL
LIN {X 0,Y 221.529,Z 261.742,A -85,B 0,C 180,E1 -20442.357,E2 -20442.357} C_VEL
LIN {X 0,Y 221.093,Z 259.988,A -85,B 0,C 180,E1 -20443.092,E2 -20443.092} C_VEL
LIN {X 0,Y 220.98,Z 259.449,A -85,B 0,C 180,E1 -20443.801,E2 -20443.801} C_VEL
LIN {X 0,Y 220.955,Z 259.458,A -85,B 0,C 180,E1 -20447.431,E2 -20447.431} C_VEL
LIN {X 0,Y 220.84,Z 259.474,A -85,B 0,C 180,E1 -20452.668,E2 -20452.668} C_VEL
LIN {X 0,Y 220.838,Z 259.477,A -85,B 0,C 180,E1 -20457.008,E2 -20457.008} C_VEL
LIN {X 0,Y 220.795,Z 259.473,A -85,B 0,C 180,E1 -20460.764,E2 -20460.764} C_VEL
LIN {X 0,Y 220.767,Z 259.463,A -85,B 0,C 180,E1 -20464.963,E2 -20464.963} C_VEL
LIN {X 0,Y 220.78,Z 259.477,A -85,B 0,C 180,E1 -20467.281,E2 -20467.281} C_VEL
LIN {X 0,Y 220.728,Z 259.465,A -85,B 0,C 180,E1 -20471.964,E2 -20471.964} C_VEL
LIN {X 0,Y 220.737,Z 259.487,A -85,B 0,C 180,E1 -20475.547,E2 -20475.547} C_VEL
LIN {X 0,Y 220.766,Z 259.453,A -85,B 0,C 180,E1 -20480.464,E2 -20480.464} C_VEL
LIN {X 0,Y 220.811,Z 259.453,A -85,B 0,C 180,E1 -20482.8,E2 -20482.8} C_VEL
LIN {X 0,Y 220.799,Z 259.476,A -85,B 0,C 180,E1 -20487.25,E2 -20487.25} C_VEL
LIN {X 0,Y 220.782,Z 259.441,A -85,B 0,C 180,E1 -20491.487,E2 -20491.487} C_VEL
LIN {X 0,Y 220.797,Z 259.477,A -85,B 0,C 180,E1 -20495.564,E2 -20495.564} C_VEL
LIN {X 0,Y 220.869,Z 259.454,A -85,B 0,C 180,E1 -20499.519,E2 -20499.519} C_VEL
LIN {X 0,Y 220.976,Z 259.413,A -85,B 0,C 180,E1 -20503.374,E2 -20503.374} C_VEL
LIN {X 0,Y 221,Z 259.451,A -85,B 0,C 180,E1 -20507.145,E2 -20507.145} C_VEL
LIN {X 0,Y 221.194,Z 259.416,A -85,B 0,C 180,E1 -20510.866,E2 -20510.866} C_VEL
LIN {X 0,Y 221.238,Z 259.386,A -85,B 0,C 180,E1 -20512.706,E2 -20512.706} C_VEL
LIN {X 0,Y 221.47,Z 259.389,A -85,B 0,C 180,E1 -20518.188,E2 -20518.188} C_VEL
LIN {X 0,Y 221.471,Z 259.385,A -85,B 0,C 180,E1 -20521.825,E2 -20521.825} C_VEL
LIN {X 0,Y 221.254,Z 259.398,A -85,B 0,C 180,E1 -20527.306,E2 -20527.306} C_VEL
LIN {X 0,Y 221.074,Z 259.446,A -85,B 0,C 180,E1 -20531.002,E2 -20531.002} C_VEL
LIN {X 0,Y 220.982,Z 259.424,A -85,B 0,C 180,E1 -20534.746,E2 -20534.746} C_VEL
LIN {X 0,Y 220.902,Z 259.463,A -85,B 0,C 180,E1 -20538.557,E2 -20538.557} C_VEL
LIN {X 0,Y 220.879,Z 259.449,A -85,B 0,C 180,E1 -20542.668,E2 -20542.668} C_VEL
LIN {X 0,Y 220.878,Z 259.468,A -85,B 0,C 180,E1 -20547.009,E2 -20547.009} C_VEL
LIN {X 0,Y 220.832,Z 259.457,A -85,B 0,C 180,E1 -20550.763,E2 -20550.763} C_VEL
LIN {X 0,Y 220.807,Z 259.482,A -85,B 0,C 180,E1 -20554.96,E2 -20554.96} C_VEL
LIN {X 0,Y 220.767,Z 259.47,A -85,B 0,C 180,E1 -20558.163,E2 -20558.163} C_VEL
LIN {X 0,Y 220.059,Z 259.573,A -85,B 0,C 180,E1 -20559.686,E2 -20559.686} C_VEL
LIN {X 0,Y 217.139,Z 259.924,A -85,B 0,C 180,E1 -20562.169,E2 -20562.169} C_VEL
LIN {X 0,Y 214.722,Z 260.236,A -85,B 0,C 180,E1 -20564.199,E2 -20564.199} C_VEL
LIN {X 0,Y 213.757,Z 260.353,A -85,B 0,C 180,E1 -20565.776,E2 -20565.776} C_VEL
LIN {X 0,Y 213.717,Z 260.356,A -85,B 0,C 180,E1 -20566.309,E2 -20566.309} C_VEL
LIN {X 0,Y 213.769,Z 260.429,A -85,B 0,C 180,E1 -20570.431,E2 -20570.431} C_VEL
LIN {X 0,Y 215.316,Z 266.57,A -85,B 0,C 180,E1 -20573.619,E2 -20573.619} C_VEL
LIN {X 0,Y 217.429,Z 271.408,A -85,B 0,C 180,E1 -20574.253,E2 -20574.253} C_VEL
LIN {X 0,Y 226.061,Z 291.288,A -85,B 0,C 180,E1 -20576.318,E2 -20576.318} C_VEL
LIN {X 0,Y 230.359,Z 303.134,A -85,B 0,C 180,E1 -20577.356,E2 -20577.356} C_VEL
LIN {X 0,Y 232.344,Z 317.733,A -85,B 0,C 180,E1 -20578.15,E2 -20578.15} C_VEL
LIN {X 0,Y 229.907,Z 374.868,A -85,B 0,C 180,E1 -20579.946,E2 -20579.946} C_VEL
LIN {X 0,Y 228.694,Z 388.044,A -85,B 0,C 180,E1 -20580.673,E2 -20580.673} C_VEL
LIN {X 0,Y 227.078,Z 400.638,A -85,B 0,C 180,E1 -20581.71,E2 -20581.71} C_VEL
LIN {X 0,Y 225.104,Z 412.677,A -85,B 0,C 180,E1 -20583.081,E2 -20583.081} C_VEL
LIN {X 0,Y 222.83,Z 424.194,A -85,B 0,C 180,E1 -20584.798,E2 -20584.798} C_VEL
LIN {X 0,Y 220.552,Z 434.585,A -85,B 0,C 180,E1 -20586.774,E2 -20586.774} C_VEL
LIN {X 0,Y 218.658,Z 442.998,A -85,B 0,C 180,E1 -20588.777,E2 -20588.777} C_VEL
LIN {X 0,Y 216.746,Z 450.9,A -85,B 0,C 180,E1 -20591.078,E2 -20591.078} C_VEL
LIN {X 0,Y 214.814,Z 458.528,A -85,B 0,C 180,E1 -20593.852,E2 -20593.852} C_VEL
LIN {X 0,Y 213.34,Z 464.654,A -85,B 0,C 180,E1 -20596.666,E2 -20596.666} C_VEL
LIN {X 0,Y 212.373,Z 469.496,A -85,B 0,C 180,E1 -20599.512,E2 -20599.512} C_VEL
LIN {X 0,Y 211.711,Z 473.193,A -85,B 0,C 180,E1 -20602.368,E2 -20602.368} C_VEL
LIN {X 0,Y 211.404,Z 476.346,A -85,B 0,C 180,E1 -20605.875,E2 -20605.875} C_VEL
LIN {X 0,Y 211.383,Z 477.558,A -85,B 0,C 180,E1 -20608.093,E2 -20608.093} C_VEL
LIN {X 0,Y 211.445,Z 478.181,A -85,B 0,C 180,E1 -20609.998,E2 -20609.998} C_VEL
LIN {X 0,Y 211.385,Z 478.412,A -85,B 0,C 180,E1 -20611.904,E2 -20611.904} C_VEL
LIN {X 0,Y 211.403,Z 478.137,A -85,B 0,C 180,E1 -20614.122,E2 -20614.122} C_VEL
LIN {X 0,Y 211.81,Z 476.637,A -85,B 0,C 180,E1 -20617.625,E2 -20617.625} C_VEL
LIN {X 0,Y 212.217,Z 475.263,A -85,B 0,C 180,E1 -20619.53,E2 -20619.53} C_VEL
LIN {X 0,Y 213.19,Z 472.371,A -85,B 0,C 180,E1 -20622.372,E2 -20622.372} C_VEL
LIN {X 0,Y 214.54,Z 468.464,A -85,B 0,C 180,E1 -20625.191,E2 -20625.191} C_VEL
LIN {X 0,Y 216.553,Z 463.444,A -85,B 0,C 180,E1 -20627.956,E2 -20627.956} C_VEL
LIN {X 0,Y 218.94,Z 457.166,A -85,B 0,C 180,E1 -20630.675,E2 -20630.675} C_VEL
LIN {X 0,Y 221.598,Z 449.629,A -85,B 0,C 180,E1 -20633.255,E2 -20633.255} C_VEL
LIN {X 0,Y 224.367,Z 441.377,A -85,B 0,C 180,E1 -20635.51,E2 -20635.51} C_VEL
LIN {X 0,Y 227.504,Z 431.684,A -85,B 0,C 180,E1 -20637.603,E2 -20637.603} C_VEL
LIN {X 0,Y 230.534,Z 420.941,A -85,B 0,C 180,E1 -20639.443,E2 -20639.443} C_VEL
LIN {X 0,Y 233.492,Z 408.742,A -85,B 0,C 180,E1 -20641.026,E2 -20641.026} C_VEL
LIN {X 0,Y 235.967,Z 395.771,A -85,B 0,C 180,E1 -20642.291,E2 -20642.291} C_VEL
LIN {X 0,Y 237.768,Z 383.154,A -85,B 0,C 180,E1 -20643.148,E2 -20643.148} C_VEL
LIN {X 0,Y 239.058,Z 370.118,A -85,B 0,C 180,E1 -20643.702,E2 -20643.702} C_VEL
LIN {X 0,Y 241.521,Z 319.655,A -85,B 0,C 180,E1 -20645.249,E2 -20645.249} C_VEL
LIN {X 0,Y 240.49,Z 312.931,A -85,B 0,C 180,E1 -20645.73,E2 -20645.73} C_VEL
LIN {X 0,Y 235.162,Z 300.394,A -85,B 0,C 180,E1 -20647.392,E2 -20647.392} C_VEL
LIN {X 0,Y 229.573,Z 289.1,A -85,B 0,C 180,E1 -20649.197,E2 -20649.197} C_VEL
LIN {X 0,Y 224.188,Z 279.625,A -85,B 0,C 180,E1 -20651.034,E2 -20651.034} C_VEL
LIN {X 0,Y 221.253,Z 274.975,A -85,B 0,C 180,E1 -20652.095,E2 -20652.095} C_VEL
LIN {X 0,Y 217.868,Z 269.752,A -85,B 0,C 180,E1 -20653.376,E2 -20653.376} C_VEL
LIN {X 0,Y 215.257,Z 265.468,A -85,B 0,C 180,E1 -20654.541,E2 -20654.541} C_VEL
LIN {X 0,Y 213.737,Z 260.47,A -85,B 0,C 180,E1 -20658.088,E2 -20658.088} C_VEL
LIN {X 0,Y 213.722,Z 260.356,A -85,B 0,C 180,E1 -20662.109,E2 -20662.109} C_VEL
LIN {X 0,Y 213.758,Z 260.354,A -85,B 0,C 180,E1 -20666.012,E2 -20666.012} C_VEL
LIN {X 0,Y 213.754,Z 260.359,A -85,B 0,C 180,E1 -20670.444,E2 -20670.444} C_VEL
LIN {X 0,Y 213.784,Z 260.355,A -85,B 0,C 180,E1 -20674.693,E2 -20674.693} C_VEL
LIN {X 0,Y 213.801,Z 260.35,A -85,B 0,C 180,E1 -20678.796,E2 -20678.796} C_VEL
LIN {X 0,Y 213.921,Z 260.327,A -85,B 0,C 180,E1 -20682.796,E2 -20682.796} C_VEL
LIN {X 0,Y 213.935,Z 260.32,A -85,B 0,C 180,E1 -20686.699,E2 -20686.699} C_VEL
LIN {X 0,Y 214.131,Z 260.3,A -85,B 0,C 180,E1 -20690.549,E2 -20690.549} C_VEL
LIN {X 0,Y 214.067,Z 260.32,A -85,B 0,C 180,E1 -20694.341,E2 -20694.341} C_VEL
LIN {X 0,Y 214.395,Z 260.274,A -85,B 0,C 180,E1 -20698.115,E2 -20698.115} C_VEL
LIN {X 0,Y 214.5,Z 260.257,A -85,B 0,C 180,E1 -20699.994,E2 -20699.994} C_VEL
LIN {X 0,Y 214.068,Z 260.319,A -85,B 0,C 180,E1 -20703.758,E2 -20703.758} C_VEL
LIN {X 0,Y 214.173,Z 260.307,A -85,B 0,C 180,E1 -20707.536,E2 -20707.536} C_VEL
LIN {X 0,Y 213.981,Z 260.33,A -85,B 0,C 180,E1 -20711.358,E2 -20711.358} C_VEL
LIN {X 0,Y 213.89,Z 260.345,A -85,B 0,C 180,E1 -20715.233,E2 -20715.233} C_VEL
LIN {X 0,Y 213.8,Z 260.352,A -85,B 0,C 180,E1 -20719.184,E2 -20719.184} C_VEL
LIN {X 0,Y 213.83,Z 260.581,A -85,B 0,C 180,E1 -20721.313,E2 -20721.313} C_VEL
LIN {X 0,Y 214.323,Z 262.19,A -85,B 0,C 180,E1 -20722.3,E2 -20722.3} C_VEL
LIN {X 0,Y 217.941,Z 267.293,A -85,B 0,C 180,E1 -20723.764,E2 -20723.764} C_VEL
LIN {X 0,Y 221.995,Z 273.572,A -85,B 0,C 180,E1 -20725.294,E2 -20725.294} C_VEL
LIN {X 0,Y 227.102,Z 281.889,A -85,B 0,C 180,E1 -20727.089,E2 -20727.089} C_VEL
LIN {X 0,Y 233.263,Z 293.087,A -85,B 0,C 180,E1 -20729.107,E2 -20729.107} C_VEL
LIN {X 0,Y 238.718,Z 304.625,A -85,B 0,C 180,E1 -20730.802,E2 -20730.802} C_VEL
LIN {X 0,Y 241.912,Z 312.536,A -85,B 0,C 180,E1 -20731.786,E2 -20731.786} C_VEL
LIN {X 0,Y 238.774,Z 369.872,A -85,B 0,C 180,E1 -20733.533,E2 -20733.533} C_VEL
LIN {X 0,Y 237.393,Z 382.094,A -85,B 0,C 180,E1 -20734.165,E2 -20734.165} C_VEL
LIN {X 0,Y 235.457,Z 395.251,A -85,B 0,C 180,E1 -20735.208,E2 -20735.208} C_VEL
LIN {X 0,Y 233.079,Z 407.177,A -85,B 0,C 180,E1 -20736.509,E2 -20736.509} C_VEL
LIN {X 0,Y 230.201,Z 418.841,A -85,B 0,C 180,E1 -20738.176,E2 -20738.176} C_VEL
LIN {X 0,Y 227.484,Z 428.367,A -85,B 0,C 180,E1 -20739.909,E2 -20739.909} C_VEL
LIN {X 0,Y 224.522,Z 437.518,A -85,B 0,C 180,E1 -20741.979,E2 -20741.979} C_VEL
LIN {X 0,Y 221.812,Z 445.291,A -85,B 0,C 180,E1 -20744.181,E2 -20744.181} C_VEL
LIN {X 0,Y 218.945,Z 453.12,A -85,B 0,C 180,E1 -20746.994,E2 -20746.994} C_VEL
LIN {X 0,Y 216.718,Z 458.785,A -85,B 0,C 180,E1 -20749.567,E2 -20749.567} C_VEL
LIN {X 0,Y 214.629,Z 464.136,A -85,B 0,C 180,E1 -20752.717,E2 -20752.717} C_VEL
LIN {X 0,Y 213.084,Z 468.079,A -85,B 0,C 180,E1 -20755.898,E2 -20755.898} C_VEL
LIN {X 0,Y 211.904,Z 471.001,A -85,B 0,C 180,E1 -20759.561,E2 -20759.561} C_VEL
LIN {X 0,Y 211.31,Z 472.201,A -85,B 0,C 180,E1 -20762.251,E2 -20762.251} C_VEL
LIN {X 0,Y 211.069,Z 472.566,A -85,B 0,C 180,E1 -20764.353,E2 -20764.353} C_VEL
LIN {X 0,Y 210.912,Z 472.487,A -85,B 0,C 180,E1 -20766.432,E2 -20766.432} C_VEL
LIN {X 0,Y 210.97,Z 471.754,A -85,B 0,C 180,E1 -20768.846,E2 -20768.846} C_VEL
LIN {X 0,Y 211.375,Z 469.388,A -85,B 0,C 180,E1 -20772.59,E2 -20772.59} C_VEL
LIN {X 0,Y 212.054,Z 466.248,A -85,B 0,C 180,E1 -20775.609,E2 -20775.609} C_VEL
LIN {X 0,Y 212.957,Z 461.977,A -85,B 0,C 180,E1 -20778.581,E2 -20778.581} C_VEL
LIN {X 0,Y 214.266,Z 456.444,A -85,B 0,C 180,E1 -20781.514,E2 -20781.514} C_VEL
LIN {X 0,Y 215.976,Z 449.484,A -85,B 0,C 180,E1 -20784.399,E2 -20784.399} C_VEL
LIN {X 0,Y 218.103,Z 441.018,A -85,B 0,C 180,E1 -20787.167,E2 -20787.167} C_VEL
LIN {X 0,Y 220.301,Z 431.779,A -85,B 0,C 180,E1 -20789.545,E2 -20789.545} C_VEL
LIN {X 0,Y 222.524,Z 421.85,A -85,B 0,C 180,E1 -20791.585,E2 -20791.585} C_VEL
LIN {X 0,Y 224.747,Z 410.935,A -85,B 0,C 180,E1 -20793.363,E2 -20793.363} C_VEL
LIN {X 0,Y 226.614,Z 399.879,A -85,B 0,C 180,E1 -20794.768,E2 -20794.768} C_VEL
LIN {X 0,Y 228.253,Z 387.381,A -85,B 0,C 180,E1 -20795.966,E2 -20795.966} C_VEL
LIN {X 0,Y 229.561,Z 374.711,A -85,B 0,C 180,E1 -20796.815,E2 -20796.815} C_VEL
LIN {X 0,Y 230.436,Z 361.254,A -85,B 0,C 180,E1 -20797.362,E2 -20797.362} C_VEL
LIN {X 0,Y 232.7,Z 305.575,A -85,B 0,C 180,E1 -20799.075,E2 -20799.075} C_VEL
LIN {X 0,Y 230.816,Z 299.691,A -85,B 0,C 180,E1 -20799.539,E2 -20799.539} C_VEL
LIN {X 0,Y 223.322,Z 280.865,A -85,B 0,C 180,E1 -20801.294,E2 -20801.294} C_VEL
LIN {X 0,Y 215.774,Z 264.971,A -85,B 0,C 180,E1 -20803.095,E2 -20803.095} C_VEL
LIN {X 0,Y 214.225,Z 261.642,A -85,B 0,C 180,E1 -20803.58,E2 -20803.58} C_VEL
LIN {X 0,Y 213.941,Z 260.426,A -85,B 0,C 180,E1 -20804.265,E2 -20804.265} C_VEL
LIN {X 0,Y 213.904,Z 260.339,A -85,B 0,C 180,E1 -20807.697,E2 -20807.697} C_VEL
LIN {X 0,Y 213.776,Z 260.347,A -85,B 0,C 180,E1 -20813.237,E2 -20813.237} C_VEL
LIN {X 0,Y 213.76,Z 260.354,A -85,B 0,C 180,E1 -20817.432,E2 -20817.432} C_VEL
LIN {X 0,Y 213.735,Z 260.361,A -85,B 0,C 180,E1 -20821.745,E2 -20821.745} C_VEL
LIN {X 0,Y 213.718,Z 260.345,A -85,B 0,C 180,E1 -20826.295,E2 -20826.295} C_VEL
LIN {X 0,Y 213.677,Z 260.35,A -85,B 0,C 180,E1 -20831.135,E2 -20831.135} C_VEL
LIN {X 0,Y 213.683,Z 260.345,A -85,B 0,C 180,E1 -20833.686,E2 -20833.686} C_VEL
LIN {X 0,Y 213.684,Z 260.367,A -85,B 0,C 180,E1 -20836.352,E2 -20836.352} C_VEL
LIN {X 0,Y 213.688,Z 260.349,A -85,B 0,C 180,E1 -20839.154,E2 -20839.154} C_VEL
LIN {X 0,Y 213.728,Z 260.345,A -85,B 0,C 180,E1 -20843.718,E2 -20843.718} C_VEL
LIN {X 0,Y 213.747,Z 260.346,A -85,B 0,C 180,E1 -20848.268,E2 -20848.268} C_VEL
LIN {X 0,Y 213.757,Z 260.321,A -85,B 0,C 180,E1 -20852.602,E2 -20852.602} C_VEL
LIN {X 0,Y 213.79,Z 260.354,A -85,B 0,C 180,E1 -20856.995,E2 -20856.995} C_VEL
LIN {X 0,Y 213.878,Z 260.293,A -85,B 0,C 180,E1 -20862.356,E2 -20862.356} C_VEL
LIN {X 0,Y 213.939,Z 260.33,A -85,B 0,C 180,E1 -20866.713,E2 -20866.713} C_VEL
LIN {X 0,Y 214.134,Z 260.3,A -85,B 0,C 180,E1 -20870.562,E2 -20870.562} C_VEL
LIN {X 0,Y 214.073,Z 260.27,A -85,B 0,C 180,E1 -20874.354,E2 -20874.354} C_VEL
LIN {X 0,Y 214.407,Z 260.268,A -85,B 0,C 180,E1 -20878.128,E2 -20878.128} C_VEL
LIN {X 0,Y 214.515,Z 260.264,A -85,B 0,C 180,E1 -20880.006,E2 -20880.006} C_VEL
LIN {X 0,Y 214.407,Z 260.264,A -85,B 0,C 180,E1 -20881.885,E2 -20881.885} C_VEL
LIN {X 0,Y 214.195,Z 260.28,A -85,B 0,C 180,E1 -20887.548,E2 -20887.548} C_VEL
LIN {X 0,Y 214.006,Z 260.325,A -85,B 0,C 180,E1 -20891.37,E2 -20891.37} C_VEL
LIN {X 0,Y 213.916,Z 260.302,A -85,B 0,C 180,E1 -20895.244,E2 -20895.244} C_VEL
LIN {X 0,Y 213.826,Z 260.35,A -85,B 0,C 180,E1 -20899.195,E2 -20899.195} C_VEL
LIN {X 0,Y 213.814,Z 260.323,A -85,B 0,C 180,E1 -20903.237,E2 -20903.237} C_VEL
LIN {X 0,Y 213.8,Z 260.354,A -85,B 0,C 180,E1 -20907.432,E2 -20907.432} C_VEL
LIN {X 0,Y 213.773,Z 260.336,A -85,B 0,C 180,E1 -20911.743,E2 -20911.743} C_VEL
LIN {X 0,Y 213.756,Z 260.348,A -85,B 0,C 180,E1 -20916.292,E2 -20916.292} C_VEL
LIN {X 0,Y 213.713,Z 260.358,A -85,B 0,C 180,E1 -20921.132,E2 -20921.132} C_VEL
LIN {X 0,Y 213.717,Z 260.355,A -85,B 0,C 180,E1 -20923.683,E2 -20923.683} C_VEL
LIN {X 0,Y 213.717,Z 260.356,A -85,B 0,C 180,E1 -20926.309,E2 -20926.309} C_VEL
LIN {X 0,Y 213.119,Z 260.519,A -85,B 0,C 180,E1 -20927.377,E2 -20927.377} C_VEL
LIN {X 0,Y 210.434,Z 261.475,A -85,B 0,C 180,E1 -20929.055,E2 -20929.055} C_VEL
LIN {X 0,Y 207.939,Z 263.397,A -85,B 0,C 180,E1 -20930.709,E2 -20930.709} C_VEL
LIN {X 0,Y 207.647,Z 265.09,A -85,B 0,C 180,E1 -20931.708,E2 -20931.708} C_VEL
LIN {X 0,Y 208.128,Z 266.814,A -85,B 0,C 180,E1 -20932.456,E2 -20932.456} C_VEL
LIN {X 0,Y 215.253,Z 282.265,A -85,B 0,C 180,E1 -20934.338,E2 -20934.338} C_VEL
LIN {X 0,Y 222.146,Z 299.129,A -85,B 0,C 180,E1 -20936.053,E2 -20936.053} C_VEL
LIN {X 0,Y 224.37,Z 305.669,A -85,B 0,C 180,E1 -20936.62,E2 -20936.62} C_VEL
LIN {X 0,Y 226.07,Z 318.258,A -85,B 0,C 180,E1 -20937.333,E2 -20937.333} C_VEL
LIN {X 0,Y 223.575,Z 374.567,A -85,B 0,C 180,E1 -20939.143,E2 -20939.143} C_VEL
LIN {X 0,Y 222.336,Z 387.698,A -85,B 0,C 180,E1 -20939.879,E2 -20939.879} C_VEL
LIN {X 0,Y 220.667,Z 400.355,A -85,B 0,C 180,E1 -20940.94,E2 -20940.94} C_VEL
LIN {X 0,Y 218.776,Z 411.654,A -85,B 0,C 180,E1 -20942.236,E2 -20942.236} C_VEL
LIN {X 0,Y 216.376,Z 423.336,A -85,B 0,C 180,E1 -20943.991,E2 -20943.991} C_VEL
LIN {X 0,Y 213.945,Z 433.854,A -85,B 0,C 180,E1 -20946.013,E2 -20946.013} C_VEL
LIN {X 0,Y 211.821,Z 443.193,A -85,B 0,C 180,E1 -20948.294,E2 -20948.294} C_VEL
LIN {X 0,Y 209.614,Z 451.772,A -85,B 0,C 180,E1 -20950.918,E2 -20950.918} C_VEL
LIN {X 0,Y 207.692,Z 459.233,A -85,B 0,C 180,E1 -20953.788,E2 -20953.788} C_VEL
LIN {X 0,Y 206.017,Z 466.076,A -85,B 0,C 180,E1 -20957.187,E2 -20957.187} C_VEL
LIN {X 0,Y 205.096,Z 470.575,A -85,B 0,C 180,E1 -20960.133,E2 -20960.133} C_VEL
LIN {X 0,Y 204.665,Z 472.941,A -85,B 0,C 180,E1 -20962.104,E2 -20962.104} C_VEL
LIN {X 0,Y 204.414,Z 474.872,A -85,B 0,C 180,E1 -20964.078,E2 -20964.078} C_VEL
LIN {X 0,Y 204.275,Z 476.453,A -85,B 0,C 180,E1 -20966.212,E2 -20966.212} C_VEL
LIN {X 0,Y 204.291,Z 477.402,A -85,B 0,C 180,E1 -20968.027,E2 -20968.027} C_VEL
LIN {X 0,Y 204.349,Z 478.048,A -85,B 0,C 180,E1 -20969.998,E2 -20969.998} C_VEL
LIN {X 0,Y 204.292,Z 478.301,A -85,B 0,C 180,E1 -20971.97,E2 -20971.97} C_VEL
LIN {X 0,Y 204.282,Z 478.152,A -85,B 0,C 180,E1 -20973.944,E2 -20973.944} C_VEL
LIN {X 0,Y 204.747,Z 476.617,A -85,B 0,C 180,E1 -20977.89,E2 -20977.89} C_VEL
LIN {X 0,Y 205.193,Z 475.268,A -85,B 0,C 180,E1 -20979.859,E2 -20979.859} C_VEL
LIN {X 0,Y 206.241,Z 472.431,A -85,B 0,C 180,E1 -20982.795,E2 -20982.795} C_VEL
LIN {X 0,Y 207.676,Z 468.586,A -85,B 0,C 180,E1 -20985.706,E2 -20985.706} C_VEL
LIN {X 0,Y 209.799,Z 463.63,A -85,B 0,C 180,E1 -20988.555,E2 -20988.555} C_VEL
LIN {X 0,Y 212.306,Z 457.421,A -85,B 0,C 180,E1 -20991.352,E2 -20991.352} C_VEL
LIN {X 0,Y 215.102,Z 449.993,A -85,B 0,C 180,E1 -20994.001,E2 -20994.001} C_VEL
LIN {X 0,Y 218.013,Z 441.831,A -85,B 0,C 180,E1 -20996.31,E2 -20996.31} C_VEL
LIN {X 0,Y 221.28,Z 432.247,A -85,B 0,C 180,E1 -20998.449,E2 -20998.449} C_VEL
LIN {X 0,Y 224.43,Z 421.646,A -85,B 0,C 180,E1 -21000.326,E2 -21000.326} C_VEL
LIN {X 0,Y 227.074,Z 411.446,A -85,B 0,C 180,E1 -21001.744,E2 -21001.744} C_VEL
LIN {X 0,Y 229.663,Z 399.34,A -85,B 0,C 180,E1 -21003.029,E2 -21003.029} C_VEL
LIN {X 0,Y 231.784,Z 386.034,A -85,B 0,C 180,E1 -21004.053,E2 -21004.053} C_VEL
LIN {X 0,Y 233.19,Z 373.81,A -85,B 0,C 180,E1 -21004.669,E2 -21004.669} C_VEL
LIN {X 0,Y 236.088,Z 320.765,A -85,B 0,C 180,E1 -21006.324,E2 -21006.324} C_VEL
LIN {X 0,Y 235.356,Z 315.883,A -85,B 0,C 180,E1 -21006.688,E2 -21006.688} C_VEL
LIN {X 0,Y 229.915,Z 303.118,A -85,B 0,C 180,E1 -21008.476,E2 -21008.476} C_VEL
LIN {X 0,Y 225.04,Z 293.148,A -85,B 0,C 180,E1 -21010.161,E2 -21010.161} C_VEL
LIN {X 0,Y 219.889,Z 283.929,A -85,B 0,C 180,E1 -21012.026,E2 -21012.026} C_VEL
LIN {X 0,Y 214.629,Z 275.485,A -85,B 0,C 180,E1 -21014.075,E2 -21014.075} C_VEL
LIN {X 0,Y 210.957,Z 270.09,A -85,B 0,C 180,E1 -21015.597,E2 -21015.597} C_VEL
LIN {X 0,Y 207.938,Z 265.356,A -85,B 0,C 180,E1 -21017.1,E2 -21017.1} C_VEL
LIN {X 0,Y 206.687,Z 261.561,A -85,B 0,C 180,E1 -21019.985,E2 -21019.985} C_VEL
LIN {X 0,Y 206.638,Z 261.241,A -85,B 0,C 180,E1 -21020.68,E2 -21020.68} C_VEL
LIN {X 0,Y 206.705,Z 261.228,A -85,B 0,C 180,E1 -21024.683,E2 -21024.683} C_VEL
LIN {X 0,Y 206.699,Z 261.229,A -85,B 0,C 180,E1 -21029.329,E2 -21029.329} C_VEL
LIN {X 0,Y 206.707,Z 261.228,A -85,B 0,C 180,E1 -21033.762,E2 -21033.762} C_VEL
LIN {X 0,Y 206.735,Z 261.222,A -85,B 0,C 180,E1 -21038.034,E2 -21038.034} C_VEL
LIN {X 0,Y 206.868,Z 261.202,A -85,B 0,C 180,E1 -21042.19,E2 -21042.19} C_VEL
LIN {X 0,Y 206.877,Z 261.2,A -85,B 0,C 180,E1 -21046.237,E2 -21046.237} C_VEL
LIN {X 0,Y 207.076,Z 261.181,A -85,B 0,C 180,E1 -21050.223,E2 -21050.223} C_VEL
LIN {X 0,Y 207.031,Z 261.197,A -85,B 0,C 180,E1 -21054.148,E2 -21054.148} C_VEL
LIN {X 0,Y 207.335,Z 261.153,A -85,B 0,C 180,E1 -21058.051,E2 -21058.051} C_VEL
LIN {X 0,Y 207.467,Z 261.132,A -85,B 0,C 180,E1 -21059.993,E2 -21059.993} C_VEL
LIN {X 0,Y 207.014,Z 261.197,A -85,B 0,C 180,E1 -21063.887,E2 -21063.887} C_VEL
LIN {X 0,Y 207.117,Z 261.187,A -85,B 0,C 180,E1 -21067.794,E2 -21067.794} C_VEL
LIN {X 0,Y 206.905,Z 261.215,A -85,B 0,C 180,E1 -21071.752,E2 -21071.752} C_VEL
LIN {X 0,Y 206.817,Z 261.223,A -85,B 0,C 180,E1 -21075.767,E2 -21075.767} C_VEL
LIN {X 0,Y 206.794,Z 261.453,A -85,B 0,C 180,E1 -21079.186,E2 -21079.186} C_VEL
LIN {X 0,Y 207.019,Z 262.446,A -85,B 0,C 180,E1 -21079.696,E2 -21079.696} C_VEL
LIN {X 0,Y 208.519,Z 265.074,A -85,B 0,C 180,E1 -21080.46,E2 -21080.46} C_VEL
LIN {X 0,Y 211.005,Z 267.899,A -85,B 0,C 180,E1 -21081.538,E2 -21081.538} C_VEL
LIN {X 0,Y 215.162,Z 273.962,A -85,B 0,C 180,E1 -21083.26,E2 -21083.26} C_VEL
LIN {X 0,Y 218.792,Z 279.582,A -85,B 0,C 180,E1 -21084.674,E2 -21084.674} C_VEL
LIN {X 0,Y 224.988,Z 290.074,A -85,B 0,C 180,E1 -21086.925,E2 -21086.925} C_VEL
LIN {X 0,Y 230.953,Z 301.786,A -85,B 0,C 180,E1 -21088.957,E2 -21088.957} C_VEL
LIN {X 0,Y 235.996,Z 313.495,A -85,B 0,C 180,E1 -21090.592,E2 -21090.592} C_VEL
LIN {X 0,Y 236.424,Z 314.581,A -85,B 0,C 180,E1 -21090.73,E2 -21090.73} C_VEL
LIN {X 0,Y 233.291,Z 369.527,A -85,B 0,C 180,E1 -21092.432,E2 -21092.432} C_VEL
LIN {X 0,Y 231.772,Z 382.509,A -85,B 0,C 180,E1 -21093.114,E2 -21093.114} C_VEL
LIN {X 0,Y 229.926,Z 394.495,A -85,B 0,C 180,E1 -21094.074,E2 -21094.074} C_VEL
LIN {X 0,Y 227.431,Z 406.763,A -85,B 0,C 180,E1 -21095.413,E2 -21095.413} C_VEL
LIN {X 0,Y 224.51,Z 418.109,A -85,B 0,C 180,E1 -21097.04,E2 -21097.04} C_VEL
LIN {X 0,Y 221.516,Z 428.233,A -85,B 0,C 180,E1 -21098.897,E2 -21098.897} C_VEL
LIN {X 0,Y 218.526,Z 437.043,A -85,B 0,C 180,E1 -21100.909,E2 -21100.909} C_VEL
LIN {X 0,Y 215.174,Z 446.158,A -85,B 0,C 180,E1 -21103.565,E2 -21103.565} C_VEL
LIN {X 0,Y 212.102,Z 454.063,A -85,B 0,C 180,E1 -21106.544,E2 -21106.544} C_VEL
LIN {X 0,Y 209.778,Z 459.601,A -85,B 0,C 180,E1 -21109.212,E2 -21109.212} C_VEL
LIN {X 0,Y 207.611,Z 464.777,A -85,B 0,C 180,E1 -21112.461,E2 -21112.461} C_VEL
LIN {X 0,Y 206.422,Z 467.556,A -85,B 0,C 180,E1 -21114.783,E2 -21114.783} C_VEL
LIN {X 0,Y 205.598,Z 469.518,A -85,B 0,C 180,E1 -21116.846,E2 -21116.846} C_VEL
LIN {X 0,Y 204.929,Z 471.036,A -85,B 0,C 180,E1 -21119.043,E2 -21119.043} C_VEL
LIN {X 0,Y 204.381,Z 472.068,A -85,B 0,C 180,E1 -21121.224,E2 -21121.224} C_VEL
LIN {X 0,Y 204.018,Z 472.626,A -85,B 0,C 180,E1 -21123.573,E2 -21123.573} C_VEL
LIN {X 0,Y 203.845,Z 472.649,A -85,B 0,C 180,E1 -21125.563,E2 -21125.563} C_VEL
LIN {X 0,Y 203.881,Z 471.954,A -85,B 0,C 180,E1 -21128.524,E2 -21128.524} C_VEL
LIN {X 0,Y 204.156,Z 470.005,A -85,B 0,C 180,E1 -21131.953,E2 -21131.953} C_VEL
LIN {X 0,Y 204.82,Z 467.066,A -85,B 0,C 180,E1 -21135.117,E2 -21135.117} C_VEL
LIN {X 0,Y 205.706,Z 463.087,A -85,B 0,C 180,E1 -21138.173,E2 -21138.173} C_VEL
LIN {X 0,Y 207.046,Z 457.597,A -85,B 0,C 180,E1 -21141.353,E2 -21141.353} C_VEL
LIN {X 0,Y 208.658,Z 451.254,A -85,B 0,C 180,E1 -21144.202,E2 -21144.202} C_VEL
LIN {X 0,Y 210.684,Z 443.434,A -85,B 0,C 180,E1 -21146.976,E2 -21146.976} C_VEL
LIN {X 0,Y 212.937,Z 434.411,A -85,B 0,C 180,E1 -21149.529,E2 -21149.529} C_VEL
LIN {X 0,Y 215.246,Z 425.048,A -85,B 0,C 180,E1 -21151.639,E2 -21151.639} C_VEL
LIN {X 0,Y 217.453,Z 414.854,A -85,B 0,C 180,E1 -21153.476,E2 -21153.476} C_VEL
LIN {X 0,Y 219.679,Z 402.678,A -85,B 0,C 180,E1 -21155.184,E2 -21155.184} C_VEL
LIN {X 0,Y 221.461,Z 390.377,A -85,B 0,C 180,E1 -21156.493,E2 -21156.493} C_VEL
LIN {X 0,Y 222.964,Z 377.157,A -85,B 0,C 180,E1 -21157.467,E2 -21157.467} C_VEL
LIN {X 0,Y 224.002,Z 363.405,A -85,B 0,C 180,E1 -21158.095,E2 -21158.095} C_VEL
LIN {X 0,Y 226.382,Z 306.527,A -85,B 0,C 180,E1 -21159.895,E2 -21159.895} C_VEL
LIN {X 0,Y 218.107,Z 285.061,A -85,B 0,C 180,E1 -21161.927,E2 -21161.927} C_VEL
LIN {X 0,Y 210.639,Z 269.137,A -85,B 0,C 180,E1 -21163.795,E2 -21163.795} C_VEL
LIN {X 0,Y 207.988,Z 264.277,A -85,B 0,C 180,E1 -21164.462,E2 -21164.462} C_VEL
LIN {X 0,Y 206.97,Z 261.85,A -85,B 0,C 180,E1 -21164.882,E2 -21164.882} C_VEL
LIN {X 0,Y 206.872,Z 261.309,A -85,B 0,C 180,E1 -21165.267,E2 -21165.267} C_VEL
LIN {X 0,Y 206.83,Z 261.222,A -85,B 0,C 180,E1 -21167.958,E2 -21167.958} C_VEL
LIN {X 0,Y 206.719,Z 261.225,A -85,B 0,C 180,E1 -21173.394,E2 -21173.394} C_VEL
LIN {X 0,Y 206.662,Z 261.227,A -85,B 0,C 180,E1 -21178.433,E2 -21178.433} C_VEL
LIN {X 0,Y 206.669,Z 261.238,A -85,B 0,C 180,E1 -21182.965,E2 -21182.965} C_VEL
LIN {X 0,Y 206.678,Z 261.217,A -85,B 0,C 180,E1 -21185.317,E2 -21185.317} C_VEL
LIN {X 0,Y 206.627,Z 261.238,A -85,B 0,C 180,E1 -21190.261,E2 -21190.261} C_VEL
LIN {X 0,Y 206.611,Z 261.233,A -85,B 0,C 180,E1 -21194.423,E2 -21194.423} C_VEL
LIN {X 0,Y 206.616,Z 261.237,A -85,B 0,C 180,E1 -21198.447,E2 -21198.447} C_VEL
LIN {X 0,Y 206.653,Z 261.21,A -85,B 0,C 180,E1 -21202.264,E2 -21202.264} C_VEL
LIN {X 0,Y 206.682,Z 261.236,A -85,B 0,C 180,E1 -21207.049,E2 -21207.049} C_VEL
LIN {X 0,Y 206.669,Z 261.197,A -85,B 0,C 180,E1 -21211.579,E2 -21211.579} C_VEL
LIN {X 0,Y 206.721,Z 261.234,A -85,B 0,C 180,E1 -21216.629,E2 -21216.629} C_VEL
LIN {X 0,Y 206.818,Z 261.172,A -85,B 0,C 180,E1 -21222.199,E2 -21222.199} C_VEL
LIN {X 0,Y 206.879,Z 261.204,A -85,B 0,C 180,E1 -21226.251,E2 -21226.251} C_VEL
LIN {X 0,Y 207.078,Z 261.18,A -85,B 0,C 180,E1 -21230.237,E2 -21230.237} C_VEL
LIN {X 0,Y 207.037,Z 261.145,A -85,B 0,C 180,E1 -21234.162,E2 -21234.162} C_VEL
LIN {X 0,Y 207.346,Z 261.147,A -85,B 0,C 180,E1 -21238.064,E2 -21238.064} C_VEL
LIN {X 0,Y 207.483,Z 261.139,A -85,B 0,C 180,E1 -21240.007,E2 -21240.007} C_VEL
LIN {X 0,Y 207.347,Z 261.142,A -85,B 0,C 180,E1 -21241.949,E2 -21241.949} C_VEL
LIN {X 0,Y 207.139,Z 261.163,A -85,B 0,C 180,E1 -21247.806,E2 -21247.806} C_VEL
LIN {X 0,Y 206.93,Z 261.206,A -85,B 0,C 180,E1 -21251.764,E2 -21251.764} C_VEL
LIN {X 0,Y 206.842,Z 261.183,A -85,B 0,C 180,E1 -21255.779,E2 -21255.779} C_VEL
LIN {X 0,Y 206.762,Z 261.23,A -85,B 0,C 180,E1 -21259.878,E2 -21259.878} C_VEL
LIN {X 0,Y 206.75,Z 261.2,A -85,B 0,C 180,E1 -21264.08,E2 -21264.08} C_VEL
LIN {X 0,Y 206.702,Z 261.238,A -85,B 0,C 180,E1 -21268.431,E2 -21268.431} C_VEL
LIN {X 0,Y 206.708,Z 261.225,A -85,B 0,C 180,E1 -21272.963,E2 -21272.963} C_VEL
LIN {X 0,Y 206.682,Z 261.223,A -85,B 0,C 180,E1 -21277.746,E2 -21277.746} C_VEL
LIN {X 0,Y 206.646,Z 261.234,A -85,B 0,C 180,E1 -21281.562,E2 -21281.562} C_VEL
LIN {X 0,Y 206.622,Z 261.24,A -85,B 0,C 180,E1 -21286.304,E2 -21286.304} C_VEL
LIN {X 0,Y 206.723,Z 261.413,A -85,B 0,C 180,E1 -21289.696,E2 -21289.696} C_VEL
LIN {X 0,Y 207.647,Z 265.09,A -85,B 0,C 180,E1 -21291.708,E2 -21291.708} C_VEL
LIN {X 0,Y 208.349,Z 267.148,A -85,B 0,C 180,E1 -21292.371,E2 -21292.371} C_VEL
LIN {X 0,Y 209.707,Z 271.155,A -85,B 0,C 180,E1 -21292.961,E2 -21292.961} C_VEL
LIN {X 0,Y 210.991,Z 278.233,A -85,B 0,C 180,E1 -21293.472,E2 -21293.472} C_VEL
LIN {X 0,Y 211.679,Z 286.594,A -85,B 0,C 180,E1 -21293.896,E2 -21293.896} C_VEL
LIN {X 0,Y 212.696,Z 292.596,A -85,B 0,C 180,E1 -21294.342,E2 -21294.342} C_VEL
LIN {X 0,Y 213.367,Z 294.459,A -85,B 0,C 180,E1 -21294.53,E2 -21294.53} C_VEL
LIN {X 0,Y 218.29,Z 307.604,A -85,B 0,C 180,E1 -21295.813,E2 -21295.813} C_VEL
LIN {X 0,Y 219.796,Z 319.564,A -85,B 0,C 180,E1 -21296.499,E2 -21296.499} C_VEL
LIN {X 0,Y 217.235,Z 374.812,A -85,B 0,C 180,E1 -21298.324,E2 -21298.324} C_VEL
LIN {X 0,Y 215.842,Z 388.788,A -85,B 0,C 180,E1 -21299.146,E2 -21299.146} C_VEL
LIN {X 0,Y 214.126,Z 401.114,A -85,B 0,C 180,E1 -21300.234,E2 -21300.234} C_VEL
LIN {X 0,Y 212.168,Z 412.183,A -85,B 0,C 180,E1 -21301.563,E2 -21301.563} C_VEL
LIN {X 0,Y 209.677,Z 423.75,A -85,B 0,C 180,E1 -21303.363,E2 -21303.363} C_VEL
LIN {X 0,Y 207.174,Z 434.184,A -85,B 0,C 180,E1 -21305.444,E2 -21305.444} C_VEL
LIN {X 0,Y 204.936,Z 443.568,A -85,B 0,C 180,E1 -21307.836,E2 -21307.836} C_VEL
LIN {X 0,Y 202.903,Z 451.27,A -85,B 0,C 180,E1 -21310.261,E2 -21310.261} C_VEL
LIN {X 0,Y 200.828,Z 458.801,A -85,B 0,C 180,E1 -21313.218,E2 -21313.218} C_VEL
LIN {X 0,Y 199.069,Z 465.738,A -85,B 0,C 180,E1 -21316.732,E2 -21316.732} C_VEL
LIN {X 0,Y 198.067,Z 470.294,A -85,B 0,C 180,E1 -21319.779,E2 -21319.779} C_VEL
LIN {X 0,Y 197.614,Z 472.686,A -85,B 0,C 180,E1 -21321.82,E2 -21321.82} C_VEL
LIN {X 0,Y 197.356,Z 474.642,A -85,B 0,C 180,E1 -21323.866,E2 -21323.866} C_VEL
LIN {X 0,Y 197.165,Z 476.517,A -85,B 0,C 180,E1 -21326.52,E2 -21326.52} C_VEL
LIN {X 0,Y 197.256,Z 477.913,A -85,B 0,C 180,E1 -21329.998,E2 -21329.998} C_VEL
LIN {X 0,Y 197.185,Z 478.127,A -85,B 0,C 180,E1 -21333.576,E2 -21333.576} C_VEL
LIN {X 0,Y 197.372,Z 477.541,A -85,B 0,C 180,E1 -21336.13,E2 -21336.13} C_VEL
LIN {X 0,Y 198.191,Z 475.285,A -85,B 0,C 180,E1 -21340.211,E2 -21340.211} C_VEL
LIN {X 0,Y 199.292,Z 472.501,A -85,B 0,C 180,E1 -21343.249,E2 -21343.249} C_VEL
LIN {X 0,Y 200.83,Z 468.712,A -85,B 0,C 180,E1 -21346.256,E2 -21346.256} C_VEL
LIN {X 0,Y 203.078,Z 463.816,A -85,B 0,C 180,E1 -21349.192,E2 -21349.192} C_VEL
LIN {X 0,Y 205.687,Z 457.674,A -85,B 0,C 180,E1 -21352.075,E2 -21352.075} C_VEL
LIN {X 0,Y 208.76,Z 450.068,A -85,B 0,C 180,E1 -21354.884,E2 -21354.884} C_VEL
LIN {X 0,Y 211.69,Z 442.319,A -85,B 0,C 180,E1 -21357.159,E2 -21357.159} C_VEL
LIN {X 0,Y 215.45,Z 431.814,A -85,B 0,C 180,E1 -21359.561,E2 -21359.561} C_VEL
LIN {X 0,Y 218.784,Z 421.163,A -85,B 0,C 180,E1 -21361.464,E2 -21361.464} C_VEL
LIN {X 0,Y 221.535,Z 410.868,A -85,B 0,C 180,E1 -21362.905,E2 -21362.905} C_VEL
LIN {X 0,Y 224.225,Z 398.582,A -85,B 0,C 180,E1 -21364.208,E2 -21364.208} C_VEL
LIN {X 0,Y 226.348,Z 385.788,A -85,B 0,C 180,E1 -21365.192,E2 -21365.192} C_VEL
LIN {X 0,Y 227.818,Z 373.476,A -85,B 0,C 180,E1 -21365.813,E2 -21365.813} C_VEL
LIN {X 0,Y 230.743,Z 321.926,A -85,B 0,C 180,E1 -21367.45,E2 -21367.45} C_VEL
LIN {X 0,Y 230.181,Z 318.682,A -85,B 0,C 180,E1 -21367.721,E2 -21367.721} C_VEL
LIN {X 0,Y 225.453,Z 307.311,A -85,B 0,C 180,E1 -21369.385,E2 -21369.385} C_VEL
LIN {X 0,Y 220.623,Z 297.247,A -85,B 0,C 180,E1 -21371.146,E2 -21371.146} C_VEL
LIN {X 0,Y 215.561,Z 288.008,A -85,B 0,C 180,E1 -21373.105,E2 -21373.105} C_VEL
LIN {X 0,Y 210.874,Z 280.481,A -85,B 0,C 180,E1 -21375.032,E2 -21375.032} C_VEL
LIN {X 0,Y 207.722,Z 275.66,A -85,B 0,C 180,E1 -21376.432,E2 -21376.432} C_VEL
LIN {X 0,Y 204.121,Z 270.338,A -85,B 0,C 180,E1 -21378.165,E2 -21378.165} C_VEL
LIN {X 0,Y 200.687,Z 265.388,A -85,B 0,C 180,E1 -21380.024,E2 -21380.024} C_VEL
LIN {X 0,Y 199.784,Z 262.885,A -85,B 0,C 180,E1 -21381.996,E2 -21381.996} C_VEL
LIN {X 0,Y 199.628,Z 262.141,A -85,B 0,C 180,E1 -21382.915,E2 -21382.915} C_VEL
LIN {X 0,Y 199.69,Z 262.101,A -85,B 0,C 180,E1 -21388.128,E2 -21388.128} C_VEL
LIN {X 0,Y 199.645,Z 262.103,A -85,B 0,C 180,E1 -21392.759,E2 -21392.759} C_VEL
LIN {X 0,Y 199.709,Z 262.094,A -85,B 0,C 180,E1 -21397.219,E2 -21397.219} C_VEL
LIN {X 0,Y 199.796,Z 262.082,A -85,B 0,C 180,E1 -21401.753,E2 -21401.753} C_VEL
LIN {X 0,Y 199.817,Z 262.081,A -85,B 0,C 180,E1 -21405.74,E2 -21405.74} C_VEL
LIN {X 0,Y 200.02,Z 262.064,A -85,B 0,C 180,E1 -21409.875,E2 -21409.875} C_VEL
LIN {X 0,Y 199.995,Z 262.074,A -85,B 0,C 180,E1 -21413.942,E2 -21413.942} C_VEL
LIN {X 0,Y 200.277,Z 262.03,A -85,B 0,C 180,E1 -21417.982,E2 -21417.982} C_VEL
LIN {X 0,Y 200.434,Z 262.008,A -85,B 0,C 180,E1 -21419.993,E2 -21419.993} C_VEL
LIN {X 0,Y 199.962,Z 262.073,A -85,B 0,C 180,E1 -21424.024,E2 -21424.024} C_VEL
LIN {X 0,Y 200.065,Z 262.064,A -85,B 0,C 180,E1 -21428.07,E2 -21428.07} C_VEL
LIN {X 0,Y 199.854,Z 262.089,A -85,B 0,C 180,E1 -21432.173,E2 -21432.173} C_VEL
LIN {X 0,Y 199.781,Z 262.201,A -85,B 0,C 180,E1 -21436.535,E2 -21436.535} C_VEL
LIN {X 0,Y 200.87,Z 265.103,A -85,B 0,C 180,E1 -21437.363,E2 -21437.363} C_VEL
LIN {X 0,Y 203.218,Z 267.374,A -85,B 0,C 180,E1 -21438.518,E2 -21438.518} C_VEL
LIN {X 0,Y 203.884,Z 268.191,A -85,B 0,C 180,E1 -21438.846,E2 -21438.846} C_VEL
LIN {X 0,Y 205.959,Z 271.362,A -85,B 0,C 180,E1 -21439.879,E2 -21439.879} C_VEL
LIN {X 0,Y 207.944,Z 273.723,A -85,B 0,C 180,E1 -21440.778,E2 -21440.778} C_VEL
LIN {X 0,Y 212.433,Z 280.518,A -85,B 0,C 180,E1 -21442.736,E2 -21442.736} C_VEL
LIN {X 0,Y 215.368,Z 285.156,A -85,B 0,C 180,E1 -21443.928,E2 -21443.928} C_VEL
LIN {X 0,Y 221.683,Z 296.266,A -85,B 0,C 180,E1 -21446.341,E2 -21446.341} C_VEL
LIN {X 0,Y 227.586,Z 308.327,A -85,B 0,C 180,E1 -21448.439,E2 -21448.439} C_VEL
LIN {X 0,Y 231.017,Z 316.711,A -85,B 0,C 180,E1 -21449.629,E2 -21449.629} C_VEL
LIN {X 0,Y 227.904,Z 369.34,A -85,B 0,C 180,E1 -21451.284,E2 -21451.284} C_VEL
LIN {X 0,Y 226.383,Z 382.055,A -85,B 0,C 180,E1 -21451.951,E2 -21451.951} C_VEL
LIN {X 0,Y 224.446,Z 394.079,A -85,B 0,C 180,E1 -21452.909,E2 -21452.909} C_VEL
LIN {X 0,Y 221.983,Z 405.952,A -85,B 0,C 180,E1 -21454.199,E2 -21454.199} C_VEL
LIN {X 0,Y 218.782,Z 417.958,A -85,B 0,C 180,E1 -21455.928,E2 -21455.928} C_VEL
LIN {X 0,Y 215.292,Z 429.219,A -85,B 0,C 180,E1 -21458.047,E2 -21458.047} C_VEL
LIN {X 0,Y 211.918,Z 438.528,A -85,B 0,C 180,E1 -21460.294,E2 -21460.294} C_VEL
LIN {X 0,Y 208.589,Z 446.954,A -85,B 0,C 180,E1 -21462.879,E2 -21462.879} C_VEL
LIN {X 0,Y 205.426,Z 454.658,A -85,B 0,C 180,E1 -21465.915,E2 -21465.915} C_VEL
LIN {X 0,Y 202.847,Z 460.402,A -85,B 0,C 180,E1 -21468.833,E2 -21468.833} C_VEL
LIN {X 0,Y 200.621,Z 465.371,A -85,B 0,C 180,E1 -21472.192,E2 -21472.192} C_VEL
LIN {X 0,Y 198.937,Z 468.98,A -85,B 0,C 180,E1 -21475.583,E2 -21475.583} C_VEL
LIN {X 0,Y 198.002,Z 471.031,A -85,B 0,C 180,E1 -21478.399,E2 -21478.399} C_VEL
LIN {X 0,Y 197.058,Z 472.58,A -85,B 0,C 180,E1 -21482.38,E2 -21482.38} C_VEL
LIN {X 0,Y 196.802,Z 472.809,A -85,B 0,C 180,E1 -21484.628,E2 -21484.628} C_VEL
LIN {X 0,Y 196.75,Z 472.136,A -85,B 0,C 180,E1 -21488.214,E2 -21488.214} C_VEL
LIN {X 0,Y 196.966,Z 470.611,A -85,B 0,C 180,E1 -21491.271,E2 -21491.271} C_VEL
LIN {X 0,Y 197.451,Z 468.507,A -85,B 0,C 180,E1 -21493.92,E2 -21493.92} C_VEL
LIN {X 0,Y 198.126,Z 465.527,A -85,B 0,C 180,E1 -21496.671,E2 -21496.671} C_VEL
LIN {X 0,Y 199.201,Z 460.985,A -85,B 0,C 180,E1 -21499.841,E2 -21499.841} C_VEL
LIN {X 0,Y 200.708,Z 455.165,A -85,B 0,C 180,E1 -21502.962,E2 -21502.962} C_VEL
LIN {X 0,Y 202.71,Z 447.827,A -85,B 0,C 180,E1 -21506.026,E2 -21506.026} C_VEL
LIN {X 0,Y 205.163,Z 438.617,A -85,B 0,C 180,E1 -21509.02,E2 -21509.02} C_VEL
LIN {X 0,Y 207.637,Z 429.104,A -85,B 0,C 180,E1 -21511.456,E2 -21511.456} C_VEL
LIN {X 0,Y 210.1,Z 418.458,A -85,B 0,C 180,E1 -21513.598,E2 -21513.598} C_VEL
LIN {X 0,Y 212.522,Z 406.747,A -85,B 0,C 180,E1 -21515.432,E2 -21515.432} C_VEL
LIN {X 0,Y 214.427,Z 395.206,A -85,B 0,C 180,E1 -21516.825,E2 -21516.825} C_VEL
LIN {X 0,Y 216.089,Z 382.376,A -85,B 0,C 180,E1 -21517.947,E2 -21517.947} C_VEL
LIN {X 0,Y 217.321,Z 369.108,A -85,B 0,C 180,E1 -21518.721,E2 -21518.721} C_VEL
LIN {X 0,Y 220.141,Z 308.193,A -85,B 0,C 180,E1 -21520.722,E2 -21520.722} C_VEL
LIN {X 0,Y 212.36,Z 288.043,A -85,B 0,C 180,E1 -21522.725,E2 -21522.725} C_VEL
LIN {X 0,Y 205.045,Z 272.434,A -85,B 0,C 180,E1 -21524.633,E2 -21524.633} C_VEL
LIN {X 0,Y 201.271,Z 265.626,A -85,B 0,C 180,E1 -21525.625,E2 -21525.625} C_VEL
LIN {X 0,Y 199.935,Z 262.897,A -85,B 0,C 180,E1 -21526.088,E2 -21526.088} C_VEL
LIN {X 0,Y 199.775,Z 262.152,A -85,B 0,C 180,E1 -21526.584,E2 -21526.584} C_VEL
LIN {X 0,Y 199.653,Z 262.107,A -85,B 0,C 180,E1 -21530.612,E2 -21530.612} C_VEL
LIN {X 0,Y 199.625,Z 262.108,A -85,B 0,C 180,E1 -21534.992,E2 -21534.992} C_VEL
LIN {X 0,Y 199.583,Z 262.106,A -85,B 0,C 180,E1 -21539.539,E2 -21539.539} C_VEL
LIN {X 0,Y 199.641,Z 262.117,A -85,B 0,C 180,E1 -21542.357,E2 -21542.357} C_VEL
LIN {X 0,Y 199.596,Z 262.107,A -85,B 0,C 180,E1 -21546.771,E2 -21546.771} C_VEL
LIN {X 0,Y 199.574,Z 262.125,A -85,B 0,C 180,E1 -21549.338,E2 -21549.338} C_VEL
LIN {X 0,Y 199.546,Z 262.1,A -85,B 0,C 180,E1 -21552.313,E2 -21552.313} C_VEL
LIN {X 0,Y 199.558,Z 262.119,A -85,B 0,C 180,E1 -21555.234,E2 -21555.234} C_VEL
LIN {X 0,Y 199.555,Z 262.122,A -85,B 0,C 180,E1 -21558.01,E2 -21558.01} C_VEL
LIN {X 0,Y 199.582,Z 262.087,A -85,B 0,C 180,E1 -21560.78,E2 -21560.78} C_VEL
LIN {X 0,Y 199.599,Z 262.121,A -85,B 0,C 180,E1 -21565.72,E2 -21565.72} C_VEL
LIN {X 0,Y 199.674,Z 262.099,A -85,B 0,C 180,E1 -21568.142,E2 -21568.142} C_VEL
LIN {X 0,Y 199.613,Z 262.083,A -85,B 0,C 180,E1 -21572.77,E2 -21572.77} C_VEL
LIN {X 0,Y 199.688,Z 262.111,A -85,B 0,C 180,E1 -21577.231,E2 -21577.231} C_VEL
LIN {X 0,Y 199.743,Z 262.054,A -85,B 0,C 180,E1 -21581.809,E2 -21581.809} C_VEL
LIN {X 0,Y 199.815,Z 262.078,A -85,B 0,C 180,E1 -21585.754,E2 -21585.754} C_VEL
LIN {X 0,Y 200.023,Z 262.06,A -85,B 0,C 180,E1 -21589.889,E2 -21589.889} C_VEL
LIN {X 0,Y 200.001,Z 262.021,A -85,B 0,C 180,E1 -21593.956,E2 -21593.956} C_VEL
LIN {X 0,Y 200.288,Z 262.025,A -85,B 0,C 180,E1 -21597.996,E2 -21597.996} C_VEL
LIN {X 0,Y 200.451,Z 262.015,A -85,B 0,C 180,E1 -21600.007,E2 -21600.007} C_VEL
LIN {X 0,Y 199.99,Z 262.031,A -85,B 0,C 180,E1 -21604.037,E2 -21604.037} C_VEL
LIN {X 0,Y 200.09,Z 262.045,A -85,B 0,C 180,E1 -21608.083,E2 -21608.083} C_VEL
LIN {X 0,Y 199.879,Z 262.078,A -85,B 0,C 180,E1 -21612.186,E2 -21612.186} C_VEL
LIN {X 0,Y 199.779,Z 262.066,A -85,B 0,C 180,E1 -21616.352,E2 -21616.352} C_VEL
LIN {X 0,Y 199.685,Z 262.11,A -85,B 0,C 180,E1 -21620.614,E2 -21620.614} C_VEL
LIN {X 0,Y 199.663,Z 262.086,A -85,B 0,C 180,E1 -21624.992,E2 -21624.992} C_VEL
LIN {X 0,Y 199.622,Z 262.109,A -85,B 0,C 180,E1 -21629.538,E2 -21629.538} C_VEL
LIN {X 0,Y 199.679,Z 262.094,A -85,B 0,C 180,E1 -21632.356,E2 -21632.356} C_VEL
LIN {X 0,Y 199.632,Z 262.103,A -85,B 0,C 180,E1 -21636.768,E2 -21636.768} C_VEL
LIN {X 0,Y 199.61,Z 262.117,A -85,B 0,C 180,E1 -21639.335,E2 -21639.335} C_VEL
LIN {X 0,Y 199.581,Z 262.11,A -85,B 0,C 180,E1 -21642.31,E2 -21642.31} C_VEL
LIN {X 0,Y 199.592,Z 262.121,A -85,B 0,C 180,E1 -21645.23,E2 -21645.23} C_VEL
LIN {X 0,Y 199.663,Z 262.286,A -85,B 0,C 180,E1 -21648.792,E2 -21648.792} C_VEL
LIN {X 0,Y 200.766,Z 266.502,A -85,B 0,C 180,E1 -21651.075,E2 -21651.075} C_VEL
LIN {X 0,Y 204.59,Z 274.354,A -85,B 0,C 180,E1 -21652.202,E2 -21652.202} C_VEL
LIN {X 0,Y 212.393,Z 292.017,A -85,B 0,C 180,E1 -21654.273,E2 -21654.273} C_VEL
LIN {X 0,Y 213.367,Z 294.459,A -85,B 0,C 180,E1 -21654.53,E2 -21654.53} C_VEL
LIN {X 0,Y 214.508,Z 298.023,A -85,B 0,C 180,E1 -21654.855,E2 -21654.855} C_VEL
LIN {X 0,Y 215.196,Z 303.777,A -85,B 0,C 180,E1 -21655.193,E2 -21655.193} C_VEL
LIN {X 0,Y 215.017,Z 309.702,A -85,B 0,C 180,E1 -21655.403,E2 -21655.403} C_VEL
LIN {X 0,Y 213.361,Z 326.003,A -85,B 0,C 180,E1 -21655.803,E2 -21655.803} C_VEL
LIN {X 0,Y 210.925,Z 375.1,A -85,B 0,C 180,E1 -21657.47,E2 -21657.47} C_VEL
LIN {X 0,Y 209.46,Z 388.971,A -85,B 0,C 180,E1 -21658.309,E2 -21658.309} C_VEL
LIN {X 0,Y 207.586,Z 401.702,A -85,B 0,C 180,E1 -21659.478,E2 -21659.478} C_VEL
LIN {X 0,Y 205.244,Z 414.216,A -85,B 0,C 180,E1 -21661.073,E2 -21661.073} C_VEL
LIN {X 0,Y 202.716,Z 425.396,A -85,B 0,C 180,E1 -21662.931,E2 -21662.931} C_VEL
LIN {X 0,Y 200.209,Z 435.452,A -85,B 0,C 180,E1 -21665.086,E2 -21665.086} C_VEL
LIN {X 0,Y 197.691,Z 445.248,A -85,B 0,C 180,E1 -21667.755,E2 -21667.755} C_VEL
LIN {X 0,Y 195.373,Z 453.46,A -85,B 0,C 180,E1 -21670.563,E2 -21670.563} C_VEL
LIN {X 0,Y 193.396,Z 460.542,A -85,B 0,C 180,E1 -21673.641,E2 -21673.641} C_VEL
LIN {X 0,Y 191.716,Z 467.008,A -85,B 0,C 180,E1 -21677.292,E2 -21677.292} C_VEL
LIN {X 0,Y 190.787,Z 471.246,A -85,B 0,C 180,E1 -21680.457,E2 -21680.457} C_VEL
LIN {X 0,Y 190.295,Z 474.399,A -85,B 0,C 180,E1 -21683.637,E2 -21683.637} C_VEL
LIN {X 0,Y 190.066,Z 476.555,A -85,B 0,C 180,E1 -21686.82,E2 -21686.82} C_VEL
LIN {X 0,Y 190.164,Z 477.776,A -85,B 0,C 180,E1 -21689.998,E2 -21689.998} C_VEL
LIN {X 0,Y 190.086,Z 478.076,A -85,B 0,C 180,E1 -21693.286,E2 -21693.286} C_VEL
LIN {X 0,Y 190.311,Z 477.506,A -85,B 0,C 180,E1 -21696.359,E2 -21696.359} C_VEL
LIN {X 0,Y 191.177,Z 475.301,A -85,B 0,C 180,E1 -21700.59,E2 -21700.59} C_VEL
LIN {X 0,Y 192.367,Z 472.571,A -85,B 0,C 180,E1 -21703.736,E2 -21703.736} C_VEL
LIN {X 0,Y 194.012,Z 468.844,A -85,B 0,C 180,E1 -21706.844,E2 -21706.844} C_VEL
LIN {X 0,Y 196.387,Z 464.02,A -85,B 0,C 180,E1 -21709.873,E2 -21709.873} C_VEL
LIN {X 0,Y 199.109,Z 457.963,A -85,B 0,C 180,E1 -21712.845,E2 -21712.845} C_VEL
LIN {X 0,Y 202.356,Z 450.455,A -85,B 0,C 180,E1 -21715.728,E2 -21715.728} C_VEL
LIN {X 0,Y 205.431,Z 442.812,A -85,B 0,C 180,E1 -21718.058,E2 -21718.058} C_VEL
LIN {X 0,Y 209.334,Z 432.462,A -85,B 0,C 180,E1 -21720.515,E2 -21720.515} C_VEL
LIN {X 0,Y 212.813,Z 421.961,A -85,B 0,C 180,E1 -21722.453,E2 -21722.453} C_VEL
LIN {X 0,Y 216.105,Z 410.262,A -85,B 0,C 180,E1 -21724.122,E2 -21724.122} C_VEL
LIN {X 0,Y 218.878,Z 397.825,A -85,B 0,C 180,E1 -21725.446,E2 -21725.446} C_VEL
LIN {X 0,Y 221.103,Z 384.823,A -85,B 0,C 180,E1 -21726.439,E2 -21726.439} C_VEL
LIN {X 0,Y 222.616,Z 372.216,A -85,B 0,C 180,E1 -21727.048,E2 -21727.048} C_VEL
LIN {X 0,Y 225.54,Z 323.313,A -85,B 0,C 180,E1 -21728.618,E2 -21728.618} C_VEL
LIN {X 0,Y 225.004,Z 321.079,A -85,B 0,C 180,E1 -21728.854,E2 -21728.854} C_VEL
LIN {X 0,Y 219.812,Z 308.587,A -85,B 0,C 180,E1 -21730.808,E2 -21730.808} C_VEL
LIN {X 0,Y 214.496,Z 297.889,A -85,B 0,C 180,E1 -21732.906,E2 -21732.906} C_VEL
LIN {X 0,Y 210.414,Z 290.679,A -85,B 0,C 180,E1 -21734.61,E2 -21734.61} C_VEL
LIN {X 0,Y 207.102,Z 285.278,A -85,B 0,C 180,E1 -21736.081,E2 -21736.081} C_VEL
LIN {X 0,Y 204.432,Z 281.073,A -85,B 0,C 180,E1 -21737.344,E2 -21737.344} C_VEL
LIN {X 0,Y 201.072,Z 276.013,A -85,B 0,C 180,E1 -21739.046,E2 -21739.046} C_VEL
LIN {X 0,Y 196.99,Z 270.314,A -85,B 0,C 180,E1 -21741.276,E2 -21741.276} C_VEL
LIN {X 0,Y 193.074,Z 264.871,A -85,B 0,C 180,E1 -21743.86,E2 -21743.86} C_VEL
LIN {X 0,Y 192.57,Z 263.017,A -85,B 0,C 180,E1 -21745.859,E2 -21745.859} C_VEL
LIN {X 0,Y 192.605,Z 262.989,A -85,B 0,C 180,E1 -21751.128,E2 -21751.128} C_VEL
LIN {X 0,Y 192.68,Z 262.971,A -85,B 0,C 180,E1 -21756.338,E2 -21756.338} C_VEL
LIN {X 0,Y 192.731,Z 262.962,A -85,B 0,C 180,E1 -21761.453,E2 -21761.453} C_VEL
LIN {X 0,Y 192.747,Z 262.966,A -85,B 0,C 180,E1 -21765.206,E2 -21765.206} C_VEL
LIN {X 0,Y 192.943,Z 262.949,A -85,B 0,C 180,E1 -21769.56,E2 -21769.56} C_VEL
LIN {X 0,Y 192.96,Z 262.949,A -85,B 0,C 180,E1 -21773.72,E2 -21773.72} C_VEL
LIN {X 0,Y 193.221,Z 262.908,A -85,B 0,C 180,E1 -21777.909,E2 -21777.909} C_VEL
LIN {X 0,Y 193.4,Z 262.884,A -85,B 0,C 180,E1 -21779.993,E2 -21779.993} C_VEL
LIN {X 0,Y 192.91,Z 262.949,A -85,B 0,C 180,E1 -21784.171,E2 -21784.171} C_VEL
LIN {X 0,Y 193.015,Z 262.938,A -85,B 0,C 180,E1 -21788.367,E2 -21788.367} C_VEL
LIN {X 0,Y 192.756,Z 263,A -85,B 0,C 180,E1 -21793.164,E2 -21793.164} C_VEL
LIN {X 0,Y 193.717,Z 265.762,A -85,B 0,C 180,E1 -21793.967,E2 -21793.967} C_VEL
LIN {X 0,Y 195.875,Z 268.058,A -85,B 0,C 180,E1 -21795.27,E2 -21795.27} C_VEL
LIN {X 0,Y 196.973,Z 268.841,A -85,B 0,C 180,E1 -21795.859,E2 -21795.859} C_VEL
LIN {X 0,Y 198.798,Z 271.928,A -85,B 0,C 180,E1 -21796.926,E2 -21796.926} C_VEL
LIN {X 0,Y 201.058,Z 274.291,A -85,B 0,C 180,E1 -21798.08,E2 -21798.08} C_VEL
LIN {X 0,Y 203.725,Z 277.96,A -85,B 0,C 180,E1 -21799.426,E2 -21799.426} C_VEL
LIN {X 0,Y 205.236,Z 280.057,A -85,B 0,C 180,E1 -21800.148,E2 -21800.148} C_VEL
LIN {X 0,Y 210.586,Z 288.283,A -85,B 0,C 180,E1 -21802.559,E2 -21802.559} C_VEL
LIN {X 0,Y 217.16,Z 300.07,A -85,B 0,C 180,E1 -21805.256,E2 -21805.256} C_VEL
LIN {X 0,Y 222.702,Z 311.522,A -85,B 0,C 180,E1 -21807.351,E2 -21807.351} C_VEL
LIN {X 0,Y 225.719,Z 318.885,A -85,B 0,C 180,E1 -21808.465,E2 -21808.465} C_VEL
LIN {X 0,Y 222.538,Z 369.954,A -85,B 0,C 180,E1 -21810.111,E2 -21810.111} C_VEL
LIN {X 0,Y 220.853,Z 383.18,A -85,B 0,C 180,E1 -21810.833,E2 -21810.833} C_VEL
LIN {X 0,Y 218.744,Z 395.458,A -85,B 0,C 180,E1 -21811.856,E2 -21811.856} C_VEL
LIN {X 0,Y 216.193,Z 406.896,A -85,B 0,C 180,E1 -21813.155,E2 -21813.155} C_VEL
LIN {X 0,Y 212.99,Z 418.296,A -85,B 0,C 180,E1 -21814.839,E2 -21814.839} C_VEL
LIN {X 0,Y 209.676,Z 428.558,A -85,B 0,C 180,E1 -21816.797,E2 -21816.797} C_VEL
LIN {X 0,Y 206.055,Z 438.16,A -85,B 0,C 180,E1 -21819.113,E2 -21819.113} C_VEL
LIN {X 0,Y 202.53,Z 446.664,A -85,B 0,C 180,E1 -21821.752,E2 -21821.752} C_VEL
LIN {X 0,Y 199.092,Z 454.524,A -85,B 0,C 180,E1 -21824.899,E2 -21824.899} C_VEL
LIN {X 0,Y 196.081,Z 460.85,A -85,B 0,C 180,E1 -21828.231,E2 -21828.231} C_VEL
LIN {X 0,Y 193.609,Z 465.965,A -85,B 0,C 180,E1 -21831.898,E2 -21831.898} C_VEL
LIN {X 0,Y 192.401,Z 468.438,A -85,B 0,C 180,E1 -21834.239,E2 -21834.239} C_VEL
LIN {X 0,Y 191.061,Z 471.057,A -85,B 0,C 180,E1 -21837.766,E2 -21837.766} C_VEL
LIN {X 0,Y 190.146,Z 472.516,A -85,B 0,C 180,E1 -21841.285,E2 -21841.285} C_VEL
LIN {X 0,Y 189.798,Z 472.871,A -85,B 0,C 180,E1 -21843.621,E2 -21843.621} C_VEL
LIN {X 0,Y 189.63,Z 472.779,A -85,B 0,C 180,E1 -21845.943,E2 -21845.943} C_VEL
LIN {X 0,Y 189.659,Z 472.172,A -85,B 0,C 180,E1 -21848.252,E2 -21848.252} C_VEL
LIN {X 0,Y 189.776,Z 471.124,A -85,B 0,C 180,E1 -21850.533,E2 -21850.533} C_VEL
LIN {X 0,Y 190.299,Z 468.823,A -85,B 0,C 180,E1 -21853.751,E2 -21853.751} C_VEL
LIN {X 0,Y 191.168,Z 465.149,A -85,B 0,C 180,E1 -21857.259,E2 -21857.259} C_VEL
